LIN {X 0.305,Y -660.831,Z 854.604,A 0.000,B 0.000,C 90.000,E1 324.689} C_DIS
LIN {X -0.046,Y -663.452,Z 854.597,A 0.000,B 0.000,C 90.000,E1 323.497} C_DIS
LIN {X 0.038,Y -665.775,Z 854.590,A 0.000,B 0.000,C 90.000,E1 322.271} C_DIS
LIN {X 0.131,Y -668.429,Z 854.581,A 0.000,B 0.000,C 90.000,E1 320.561} C_DIS
LIN {X -0.225,Y -670.175,Z 854.573,A 0.000,B 0.000,C 90.000,E1 319.138} C_DIS
LIN {X -0.142,Y -671.073,Z 854.569,A 0.000,B 0.000,C 90.000,E1 318.405} C_DIS
LIN {X 0.016,Y -673.504,Z 854.558,A 0.000,B 0.000,C 90.000,E1 316.458} C_DIS
LIN {X 0.136,Y -674.995,Z 854.551,A 0.000,B 0.000,C 90.000,E1 315.243} C_DIS
LIN {X 0.192,Y -675.409,Z 854.549,A 0.000,B 0.000,C 90.000,E1 314.757} C_DIS
LIN {X -0.057,Y -677.144,Z 854.539,A 0.000,B 0.000,C 90.000,E1 313.095} C_DIS
LIN {X -0.311,Y -678.588,Z 854.531,A 0.000,B 0.000,C 90.000,E1 311.676} C_DIS
LIN {X -0.045,Y -679.939,Z 854.523,A 0.000,B 0.000,C 90.000,E1 310.216} C_DIS
LIN {X 0.327,Y -681.172,Z 854.516,A 0.000,B 0.000,C 90.000,E1 308.749} C_DIS
LIN {X -0.229,Y -682.419,Z 854.508,A 0.000,B 0.000,C 90.000,E1 307.363} C_DIS
LIN {X -0.224,Y -683.571,Z 854.500,A 0.000,B 0.000,C 90.000,E1 305.931} C_DIS
LIN {X -0.035,Y -684.565,Z 854.492,A 0.000,B 0.000,C 90.000,E1 304.485} C_DIS
LIN {X -0.013,Y -685.390,Z 854.485,A 0.000,B 0.000,C 90.000,E1 303.293} C_DIS
LIN {X 0.041,Y -686.764,Z 854.474,A 0.000,B 0.000,C 90.000,E1 301.386} C_DIS
LIN {X 0.019,Y -688.211,Z 854.464,A 0.000,B 0.000,C 90.000,E1 299.489} C_DIS
LIN {X -0.183,Y -689.701,Z 854.455,A 0.000,B 0.000,C 90.000,E1 297.847} C_DIS
LIN {X -0.206,Y -691.756,Z 854.443,A 0.000,B 0.000,C 90.000,E1 295.720} C_DIS
LIN {X -0.161,Y -692.641,Z 854.438,A 0.000,B 0.000,C 90.000,E1 294.771} C_DIS
LIN {X -0.106,Y -693.267,Z 854.432,A 0.000,B 0.000,C 90.000,E1 293.823} C_DIS
LIN {X 0.103,Y -693.192,Z 854.430,A 0.000,B 0.000,C 90.000,E1 293.334} C_DIS
LIN {X 0.345,Y -692.866,Z 854.428,A 0.000,B 0.000,C 90.000,E1 293.078} C_DIS
LIN {X -0.083,Y -691.503,Z 854.426,A 0.000,B 0.000,C 90.000,E1 292.642} C_DIS
LIN {X 0.153,Y -690.318,Z 854.424,A 0.000,B 0.000,C 90.000,E1 292.386} C_DIS
LIN {X 0.345,Y -685.933,Z 854.422,A 0.000,B 0.000,C 90.000,E1 291.897} C_DIS
LIN {X 0.197,Y -684.631,Z 854.421,A 0.000,B 0.000,C 90.000,E1 291.791} C_DIS
LIN {X -0.331,Y -682.554,Z 854.421,A 0.000,B 0.000,C 90.000,E1 291.716} C_DIS
LIN {X -0.153,Y -676.537,Z 854.419,A 0.000,B 0.000,C 90.000,E1 291.461} C_DIS
LIN {X -0.305,Y -674.797,Z 854.419,A 0.000,B 0.000,C 90.000,E1 291.408} C_DIS
LIN {X -0.113,Y -671.365,Z 854.418,A 0.000,B 0.000,C 90.000,E1 291.280} C_DIS
LIN {X 0.071,Y -666.701,Z 854.418,A 0.000,B 0.000,C 90.000,E1 291.153} C_DIS
LIN {X 0.182,Y -654.493,Z 854.416,A 0.000,B 0.000,C 90.000,E1 290.865} C_DIS
LIN {X -0.225,Y -651.097,Z 854.415,A 0.000,B 0.000,C 90.000,E1 290.791} C_DIS
LIN {X 0.006,Y -647.543,Z 854.415,A 0.000,B 0.000,C 90.000,E1 290.663} C_DIS
LIN {X -0.286,Y -642.427,Z 854.413,A 0.000,B 0.000,C 90.000,E1 290.429} C_DIS
LIN {X -0.345,Y -642.340,Z 854.413,A 0.000,B 0.000,C 90.000,E1 290.429} C_DIS
LIN {X 0.256,Y -640.659,Z 854.412,A 0.000,B 0.000,C 90.000,E1 290.174} C_DIS
LIN {X 0.212,Y -640.651,Z 854.412,A 0.000,B 0.000,C 90.000,E1 290.174} C_DIS
LIN {X 0.313,Y -640.504,Z 854.411,A 0.000,B 0.000,C 90.000,E1 289.993} C_DIS
LIN {X 0.066,Y -642.134,Z 854.409,A 0.000,B 0.000,C 90.000,E1 289.577} C_DIS
LIN {X -0.280,Y -649.483,Z 854.401,A 0.000,B 0.000,C 90.000,E1 288.236} C_DIS
LIN {X 0.093,Y -652.491,Z 854.398,A 0.000,B 0.000,C 90.000,E1 287.583} C_DIS
LIN {X -0.092,Y -655.744,Z 854.394,A 0.000,B 0.000,C 90.000,E1 286.858} C_DIS
LIN {X -0.254,Y -658.563,Z 854.390,A 0.000,B 0.000,C 90.000,E1 286.134} C_DIS
LIN {X 0.166,Y -660.214,Z 854.387,A 0.000,B 0.000,C 90.000,E1 285.607} C_DIS
LIN {X -0.131,Y -662.219,Z 854.383,A 0.000,B 0.000,C 90.000,E1 284.898} C_DIS
LIN {X -0.152,Y -663.344,Z 854.380,A 0.000,B 0.000,C 90.000,E1 284.411} C_DIS
LIN {X 0.134,Y -664.877,Z 854.375,A 0.000,B 0.000,C 90.000,E1 283.411} C_DIS
LIN {X -0.038,Y -665.424,Z 854.372,A 0.000,B 0.000,C 90.000,E1 282.939} C_DIS
LIN {X -0.351,Y -665.777,Z 854.369,A 0.000,B 0.000,C 90.000,E1 282.479} C_DIS
LIN {X 0.052,Y -665.985,Z 854.365,A 0.000,B 0.000,C 90.000,E1 281.715} C_DIS
LIN {X -0.115,Y -665.854,Z 854.362,A 0.000,B 0.000,C 90.000,E1 281.243} C_DIS
LIN {X 0.244,Y -665.514,Z 854.360,A 0.000,B 0.000,C 90.000,E1 280.725} C_DIS
LIN {X 0.071,Y -664.975,Z 854.357,A 0.000,B 0.000,C 90.000,E1 280.254} C_DIS
LIN {X -0.223,Y -664.156,Z 854.354,A 0.000,B 0.000,C 90.000,E1 279.792} C_DIS
LIN {X 0.244,Y -663.077,Z 854.352,A 0.000,B 0.000,C 90.000,E1 279.265} C_DIS
LIN {X -0.059,Y -661.694,Z 854.349,A 0.000,B 0.000,C 90.000,E1 278.803} C_DIS
LIN {X -0.270,Y -659.846,Z 854.346,A 0.000,B 0.000,C 90.000,E1 278.333} C_DIS
LIN {X 0.062,Y -657.762,Z 854.344,A 0.000,B 0.000,C 90.000,E1 277.814} C_DIS
LIN {X -0.164,Y -655.944,Z 854.341,A 0.000,B 0.000,C 90.000,E1 277.466} C_DIS
LIN {X 0.140,Y -653.194,Z 854.339,A 0.000,B 0.000,C 90.000,E1 276.947} C_DIS
LIN {X -0.186,Y -650.972,Z 854.337,A 0.000,B 0.000,C 90.000,E1 276.606} C_DIS
LIN {X 0.040,Y -646.524,Z 854.333,A 0.000,B 0.000,C 90.000,E1 275.967} C_DIS
LIN {X 0.214,Y -642.388,Z 854.330,A 0.000,B 0.000,C 90.000,E1 275.454} C_DIS
LIN {X -0.152,Y -637.498,Z 854.328,A 0.000,B 0.000,C 90.000,E1 274.992} C_DIS
LIN {X -0.286,Y -632.086,Z 854.325,A 0.000,B 0.000,C 90.000,E1 274.531} C_DIS
LIN {X 0.052,Y -624.823,Z 854.322,A 0.000,B 0.000,C 90.000,E1 273.955} C_DIS
LIN {X -0.171,Y -617.371,Z 854.319,A 0.000,B 0.000,C 90.000,E1 273.498} C_DIS
LIN {X 0.225,Y -611.014,Z 854.317,A 0.000,B 0.000,C 90.000,E1 273.094} C_DIS
LIN {X 0.111,Y -602.470,Z 854.315,A 0.000,B 0.000,C 90.000,E1 272.694} C_DIS
LIN {X 0.147,Y -597.447,Z 854.314,A 0.000,B 0.000,C 90.000,E1 272.465} C_DIS
LIN {X -0.262,Y -590.199,Z 854.312,A 0.000,B 0.000,C 90.000,E1 272.236} C_DIS
LIN {X -0.231,Y -584.532,Z 854.311,A 0.000,B 0.000,C 90.000,E1 272.064} C_DIS
LIN {X 0.037,Y -578.213,Z 854.311,A 0.000,B 0.000,C 90.000,E1 271.892} C_DIS
LIN {X 0.152,Y -571.643,Z 854.310,A 0.000,B 0.000,C 90.000,E1 271.776} C_DIS
LIN {X 0.073,Y -564.068,Z 854.310,A 0.000,B 0.000,C 90.000,E1 271.718} C_DIS
LIN {X -0.186,Y -556.079,Z 854.310,A 0.000,B 0.000,C 90.000,E1 271.718} C_DIS
LIN {X 0.047,Y -552.503,Z 854.309,A 0.000,B 0.000,C 90.000,E1 271.661} C_DIS
LIN {X 0.113,Y -549.285,Z 854.309,A 0.000,B 0.000,C 90.000,E1 271.547} C_DIS
LIN {X 0.107,Y -548.823,Z 854.308,A 0.000,B 0.000,C 90.000,E1 271.489} C_DIS
LIN {X -0.141,Y -548.111,Z 854.308,A 0.000,B 0.000,C 90.000,E1 271.375} C_DIS
LIN {X 0.206,Y -547.113,Z 854.305,A 0.000,B 0.000,C 90.000,E1 270.917} C_DIS
LIN {X -0.204,Y -546.071,Z 854.301,A 0.000,B 0.000,C 90.000,E1 270.115} C_DIS
LIN {X 0.156,Y -544.002,Z 854.286,A 0.000,B 0.000,C 90.000,E1 267.535} C_DIS
LIN {X -0.125,Y -542.650,Z 854.275,A 0.000,B 0.000,C 90.000,E1 265.584} C_DIS
LIN {X 0.127,Y -541.454,Z 854.266,A 0.000,B 0.000,C 90.000,E1 263.856} C_DIS
LIN {X -0.258,Y -540.437,Z 854.260,A 0.000,B 0.000,C 90.000,E1 262.761} C_DIS
LIN {X 0.069,Y -538.715,Z 854.249,A 0.000,B 0.000,C 90.000,E1 260.735} C_DIS
LIN {X -0.098,Y -536.794,Z 854.238,A 0.000,B 0.000,C 90.000,E1 258.757} C_DIS
LIN {X 0.196,Y -535.279,Z 854.230,A 0.000,B 0.000,C 90.000,E1 257.297} C_DIS
LIN {X 0.007,Y -533.945,Z 854.223,A 0.000,B 0.000,C 90.000,E1 256.172} C_DIS
LIN {X 0.098,Y -531.188,Z 854.210,A 0.000,B 0.000,C 90.000,E1 253.866} C_DIS
LIN {X 0.181,Y -529.507,Z 854.202,A 0.000,B 0.000,C 90.000,E1 252.417} C_DIS
LIN {X 0.244,Y -527.676,Z 854.194,A 0.000,B 0.000,C 90.000,E1 250.967} C_DIS
LIN {X 0.094,Y -526.170,Z 854.188,A 0.000,B 0.000,C 90.000,E1 249.826} C_DIS
LIN {X -0.227,Y -524.242,Z 854.180,A 0.000,B 0.000,C 90.000,E1 248.411} C_DIS
LIN {X -0.222,Y -521.671,Z 854.170,A 0.000,B 0.000,C 90.000,E1 246.666} C_DIS
LIN {X -0.092,Y -519.902,Z 854.164,A 0.000,B 0.000,C 90.000,E1 245.485} C_DIS
LIN {X 0.223,Y -518.082,Z 854.157,A 0.000,B 0.000,C 90.000,E1 244.280} C_DIS
LIN {X 0.046,Y -516.123,Z 854.151,A 0.000,B 0.000,C 90.000,E1 243.127} C_DIS
LIN {X 0.192,Y -512.528,Z 854.139,A 0.000,B 0.000,C 90.000,E1 241.051} C_DIS
LIN {X -0.167,Y -510.982,Z 854.134,A 0.000,B 0.000,C 90.000,E1 240.205} C_DIS
LIN {X 0.011,Y -507.628,Z 854.125,A 0.000,B 0.000,C 90.000,E1 238.408} C_DIS
LIN {X 0.062,Y -504.750,Z 854.116,A 0.000,B 0.000,C 90.000,E1 236.914} C_DIS
LIN {X 0.150,Y -502.887,Z 854.111,A 0.000,B 0.000,C 90.000,E1 236.008} C_DIS
LIN {X 0.101,Y -500.210,Z 854.105,A 0.000,B 0.000,C 90.000,E1 234.815} C_DIS
LIN {X 0.013,Y -497.365,Z 854.098,A 0.000,B 0.000,C 90.000,E1 233.623} C_DIS
LIN {X -0.105,Y -493.157,Z 854.088,A 0.000,B 0.000,C 90.000,E1 231.823} C_DIS
LIN {X -0.015,Y -488.793,Z 854.078,A 0.000,B 0.000,C 90.000,E1 229.989} C_DIS
LIN {X 0.093,Y -485.390,Z 854.069,A 0.000,B 0.000,C 90.000,E1 228.447} C_DIS
LIN {X -0.011,Y -479.194,Z 854.054,A 0.000,B 0.000,C 90.000,E1 225.688} C_DIS
LIN {X 0.233,Y -475.930,Z 854.045,A 0.000,B 0.000,C 90.000,E1 224.109} C_DIS
LIN {X 0.057,Y -470.544,Z 854.031,A 0.000,B 0.000,C 90.000,E1 221.634} C_DIS
LIN {X -0.111,Y -466.488,Z 854.021,A 0.000,B 0.000,C 90.000,E1 219.769} C_DIS
LIN {X 0.236,Y -463.871,Z 854.014,A 0.000,B 0.000,C 90.000,E1 218.463} C_DIS
LIN {X -0.220,Y -459.270,Z 854.002,A 0.000,B 0.000,C 90.000,E1 216.297} C_DIS
LIN {X -0.065,Y -454.412,Z 853.989,A 0.000,B 0.000,C 90.000,E1 214.040} C_DIS
LIN {X -0.094,Y -448.929,Z 853.975,A 0.000,B 0.000,C 90.000,E1 211.465} C_DIS
LIN {X -0.142,Y -443.436,Z 853.960,A 0.000,B 0.000,C 90.000,E1 208.871} C_DIS
LIN {X 0.082,Y -440.075,Z 853.951,A 0.000,B 0.000,C 90.000,E1 207.206} C_DIS
LIN {X -0.149,Y -436.707,Z 853.942,A 0.000,B 0.000,C 90.000,E1 205.591} C_DIS
LIN {X -0.023,Y -432.647,Z 853.931,A 0.000,B 0.000,C 90.000,E1 203.590} C_DIS
LIN {X 0.004,Y -428.619,Z 853.920,A 0.000,B 0.000,C 90.000,E1 201.589} C_DIS
LIN {X 0.020,Y -426.021,Z 853.913,A 0.000,B 0.000,C 90.000,E1 200.248} C_DIS
LIN {X 0.149,Y -421.439,Z 853.899,A 0.000,B 0.000,C 90.000,E1 197.873} C_DIS
LIN {X -0.038,Y -418.215,Z 853.890,A 0.000,B 0.000,C 90.000,E1 196.205} C_DIS
LIN {X -0.074,Y -416.086,Z 853.884,A 0.000,B 0.000,C 90.000,E1 195.190} C_DIS
LIN {X -0.103,Y -413.280,Z 853.877,A 0.000,B 0.000,C 90.000,E1 193.828} C_DIS
LIN {X 0.018,Y -407.250,Z 853.860,A 0.000,B 0.000,C 90.000,E1 190.715} C_DIS
LIN {X 0.083,Y -403.143,Z 853.848,A 0.000,B 0.000,C 90.000,E1 188.624} C_DIS
LIN {X -0.057,Y -399.072,Z 853.836,A 0.000,B 0.000,C 90.000,E1 186.549} C_DIS
LIN {X -0.128,Y -392.992,Z 853.817,A 0.000,B 0.000,C 90.000,E1 183.037} C_DIS
LIN {X 0.111,Y -389.410,Z 853.803,A 0.000,B 0.000,C 90.000,E1 180.516} C_DIS
LIN {X 0.050,Y -386.974,Z 853.793,A 0.000,B 0.000,C 90.000,E1 178.740} C_DIS
LIN {X -0.143,Y -383.971,Z 853.781,A 0.000,B 0.000,C 90.000,E1 176.617} C_DIS
LIN {X 0.096,Y -381.531,Z 853.771,A 0.000,B 0.000,C 90.000,E1 174.780} C_DIS
LIN {X 0.013,Y -377.867,Z 853.755,A 0.000,B 0.000,C 90.000,E1 171.894} C_DIS
LIN {X 0.064,Y -372.888,Z 853.725,A 0.000,B 0.000,C 90.000,E1 166.408} C_DIS
LIN {X 0.059,Y -372.070,Z 853.714,A 0.000,B 0.000,C 90.000,E1 164.574} C_DIS
LIN {X 0.138,Y -372.143,Z 853.704,A 0.000,B 0.000,C 90.000,E1 162.725} C_DIS
LIN {X 0.072,Y -372.712,Z 853.700,A 0.000,B 0.000,C 90.000,E1 162.000} C_DIS
LIN {X -0.017,Y -374.058,Z 853.694,A 0.000,B 0.000,C 90.000,E1 160.913} C_DIS
LIN {X -0.010,Y -374.593,Z 853.693,A 0.000,B 0.000,C 90.000,E1 160.678} C_DIS
LIN {X 0.068,Y -375.876,Z 853.689,A 0.000,B 0.000,C 90.000,E1 159.934} C_DIS
LIN {X 0.047,Y -376.938,Z 853.687,A 0.000,B 0.000,C 90.000,E1 159.571} C_DIS
LIN {X 0.132,Y -378.868,Z 853.684,A 0.000,B 0.000,C 90.000,E1 159.028} C_DIS
LIN {X 0.124,Y -379.696,Z 853.683,A 0.000,B 0.000,C 90.000,E1 158.847} C_DIS
LIN {X -0.100,Y -384.318,Z 853.679,A 0.000,B 0.000,C 90.000,E1 158.156} C_DIS
LIN {X 0.155,Y -385.649,Z 853.678,A 0.000,B 0.000,C 90.000,E1 157.975} C_DIS
LIN {X -0.074,Y -390.628,Z 853.675,A 0.000,B 0.000,C 90.000,E1 157.592} C_DIS
LIN {X -0.108,Y -392.245,Z 853.675,A 0.000,B 0.000,C 90.000,E1 157.486} C_DIS
LIN {X 0.020,Y -398.045,Z 853.673,A 0.000,B 0.000,C 90.000,E1 157.177} C_DIS
LIN {X -0.120,Y -408.863,Z 853.671,A 0.000,B 0.000,C 90.000,E1 156.741} C_DIS
LIN {X -0.192,Y -415.764,Z 853.669,A 0.000,B 0.000,C 90.000,E1 156.485} C_DIS
LIN {X -0.146,Y -422.411,Z 853.668,A 0.000,B 0.000,C 90.000,E1 156.177} C_DIS
LIN {X -0.191,Y -430.182,Z 853.665,A 0.000,B 0.000,C 90.000,E1 155.741} C_DIS
LIN {X -0.154,Y -438.432,Z 853.662,A 0.000,B 0.000,C 90.000,E1 155.229} C_DIS
LIN {X 0.170,Y -447.724,Z 853.659,A 0.000,B 0.000,C 90.000,E1 154.537} C_DIS
LIN {X 0.036,Y -458.604,Z 853.654,A 0.000,B 0.000,C 90.000,E1 153.691} C_DIS
LIN {X -0.049,Y -464.301,Z 853.651,A 0.000,B 0.000,C 90.000,E1 153.179} C_DIS
LIN {X -0.045,Y -469.880,Z 853.648,A 0.000,B 0.000,C 90.000,E1 152.615} C_DIS
LIN {X -0.010,Y -475.194,Z 853.645,A 0.000,B 0.000,C 90.000,E1 152.025} C_DIS
LIN {X -0.089,Y -484.388,Z 853.639,A 0.000,B 0.000,C 90.000,E1 151.001} C_DIS
LIN {X -0.014,Y -492.068,Z 853.634,A 0.000,B 0.000,C 90.000,E1 150.078} C_DIS
LIN {X 0.097,Y -499.047,Z 853.629,A 0.000,B 0.000,C 90.000,E1 149.154} C_DIS
LIN {X -0.009,Y -502.452,Z 853.626,A 0.000,B 0.000,C 90.000,E1 148.742} C_DIS
LIN {X -0.212,Y -509.109,Z 853.621,A 0.000,B 0.000,C 90.000,E1 147.867} C_DIS
LIN {X 0.286,Y -517.023,Z 853.615,A 0.000,B 0.000,C 90.000,E1 146.628} C_DIS
LIN {X -0.021,Y -521.485,Z 853.611,A 0.000,B 0.000,C 90.000,E1 145.928} C_DIS
LIN {X 0.109,Y -527.451,Z 853.605,A 0.000,B 0.000,C 90.000,E1 144.895} C_DIS
LIN {X -0.108,Y -531.445,Z 853.601,A 0.000,B 0.000,C 90.000,E1 144.196} C_DIS
LIN {X 0.087,Y -543.109,Z 853.589,A 0.000,B 0.000,C 90.000,E1 142.029} C_DIS
LIN {X -0.091,Y -552.534,Z 853.580,A 0.000,B 0.000,C 90.000,E1 140.356} C_DIS
LIN {X 0.031,Y -555.668,Z 853.577,A 0.000,B 0.000,C 90.000,E1 139.784} C_DIS
LIN {X 0.081,Y -562.213,Z 853.570,A 0.000,B 0.000,C 90.000,E1 138.528} C_DIS
LIN {X -0.024,Y -570.218,Z 853.561,A 0.000,B 0.000,C 90.000,E1 137.025} C_DIS
LIN {X 0.140,Y -574.938,Z 853.556,A 0.000,B 0.000,C 90.000,E1 136.053} C_DIS
LIN {X -0.175,Y -580.233,Z 853.550,A 0.000,B 0.000,C 90.000,E1 135.000} C_DIS
LIN {X 0.000,Y -585.465,Z 853.544,A 0.000,B 0.000,C 90.000,E1 133.905} C_DIS
LIN {X -0.065,Y -589.929,Z 853.539,A 0.000,B 0.000,C 90.000,E1 132.975} C_DIS
LIN {X 0.178,Y -592.991,Z 853.535,A 0.000,B 0.000,C 90.000,E1 132.285} C_DIS
LIN {X -0.098,Y -598.779,Z 853.528,A 0.000,B 0.000,C 90.000,E1 130.987} C_DIS
LIN {X 0.179,Y -604.404,Z 853.520,A 0.000,B 0.000,C 90.000,E1 129.644} C_DIS
LIN {X -0.033,Y -605.514,Z 853.519,A 0.000,B 0.000,C 90.000,E1 129.402} C_DIS
LIN {X -0.025,Y -610.395,Z 853.512,A 0.000,B 0.000,C 90.000,E1 128.096} C_DIS
LIN {X -0.029,Y -613.075,Z 853.507,A 0.000,B 0.000,C 90.000,E1 127.317} C_DIS
LIN {X 0.001,Y -615.649,Z 853.503,A 0.000,B 0.000,C 90.000,E1 126.537} C_DIS
LIN {X 0.180,Y -619.642,Z 853.496,A 0.000,B 0.000,C 90.000,E1 125.231} C_DIS
LIN {X -0.298,Y -623.002,Z 853.489,A 0.000,B 0.000,C 90.000,E1 123.992} C_DIS
LIN {X -0.189,Y -625.312,Z 853.483,A 0.000,B 0.000,C 90.000,E1 122.959} C_DIS
LIN {X -0.390,Y -626.894,Z 853.479,A 0.000,B 0.000,C 90.000,E1 122.212} C_DIS
LIN {X 0.298,Y -628.727,Z 853.473,A 0.000,B 0.000,C 90.000,E1 121.131} C_DIS
LIN {X 0.196,Y -631.203,Z 853.465,A 0.000,B 0.000,C 90.000,E1 119.617} C_DIS
LIN {X 0.040,Y -632.158,Z 853.460,A 0.000,B 0.000,C 90.000,E1 118.871} C_DIS
LIN {X 0.141,Y -633.050,Z 853.456,A 0.000,B 0.000,C 90.000,E1 118.103} C_DIS
LIN {X -0.267,Y -633.921,Z 853.451,A 0.000,B 0.000,C 90.000,E1 117.129} C_DIS
LIN {X -0.185,Y -634.207,Z 853.448,A 0.000,B 0.000,C 90.000,E1 116.616} C_DIS
LIN {X -0.017,Y -634.318,Z 853.442,A 0.000,B 0.000,C 90.000,E1 115.591} C_DIS
LIN {X 0.025,Y -634.254,Z 853.441,A 0.000,B 0.000,C 90.000,E1 115.335} C_DIS
LIN {X -0.078,Y -633.499,Z 853.435,A 0.000,B 0.000,C 90.000,E1 114.335} C_DIS
LIN {X -0.003,Y -632.746,Z 853.432,A 0.000,B 0.000,C 90.000,E1 113.823} C_DIS
LIN {X -0.188,Y -631.298,Z 853.430,A 0.000,B 0.000,C 90.000,E1 113.334} C_DIS
LIN {X -0.157,Y -630.372,Z 853.428,A 0.000,B 0.000,C 90.000,E1 113.078} C_DIS
LIN {X -0.144,Y -629.516,Z 853.427,A 0.000,B 0.000,C 90.000,E1 112.950} C_DIS
LIN {X -0.353,Y -627.650,Z 853.425,A 0.000,B 0.000,C 90.000,E1 112.589} C_DIS
LIN {X -0.344,Y -626.450,Z 853.425,A 0.000,B 0.000,C 90.000,E1 112.461} C_DIS
LIN {X 0.250,Y -623.409,Z 853.423,A 0.000,B 0.000,C 90.000,E1 112.025} C_DIS
LIN {X 0.248,Y -620.100,Z 853.421,A 0.000,B 0.000,C 90.000,E1 111.770} C_DIS
LIN {X 0.026,Y -617.046,Z 853.420,A 0.000,B 0.000,C 90.000,E1 111.535} C_DIS
LIN {X -0.217,Y -610.855,Z 853.417,A 0.000,B 0.000,C 90.000,E1 111.153} C_DIS
LIN {X -0.223,Y -601.454,Z 853.414,A 0.000,B 0.000,C 90.000,E1 110.610} C_DIS
LIN {X -0.157,Y -594.867,Z 853.412,A 0.000,B 0.000,C 90.000,E1 110.248} C_DIS
LIN {X 0.163,Y -588.110,Z 853.411,A 0.000,B 0.000,C 90.000,E1 109.885} C_DIS
LIN {X -0.289,Y -579.028,Z 853.409,A 0.000,B 0.000,C 90.000,E1 109.577} C_DIS
LIN {X -0.286,Y -574.865,Z 853.408,A 0.000,B 0.000,C 90.000,E1 109.450} C_DIS
LIN {X 0.034,Y -567.390,Z 853.406,A 0.000,B 0.000,C 90.000,E1 109.141} C_DIS
LIN {X -0.054,Y -566.248,Z 853.406,A 0.000,B 0.000,C 90.000,E1 109.087} C_DIS
LIN {X -0.125,Y -564.156,Z 853.405,A 0.000,B 0.000,C 90.000,E1 108.906} C_DIS
LIN {X -0.220,Y -562.671,Z 853.404,A 0.000,B 0.000,C 90.000,E1 108.671} C_DIS
LIN {X 0.137,Y -561.346,Z 853.401,A 0.000,B 0.000,C 90.000,E1 108.236} C_DIS
LIN {X 0.160,Y -560.574,Z 853.399,A 0.000,B 0.000,C 90.000,E1 107.819} C_DIS
LIN {X 0.251,Y -560.171,Z 853.394,A 0.000,B 0.000,C 90.000,E1 106.858} C_DIS
LIN {X -0.233,Y -561.442,Z 853.369,A 0.000,B 0.000,C 90.000,E1 102.479} C_DIS
LIN {X -0.084,Y -562.863,Z 853.357,A 0.000,B 0.000,C 90.000,E1 100.254} C_DIS
LIN {X 0.063,Y -563.850,Z 853.349,A 0.000,B 0.000,C 90.000,E1 98.859} C_DIS
LIN {X 0.147,Y -564.822,Z 853.342,A 0.000,B 0.000,C 90.000,E1 97.473} C_DIS
LIN {X -0.153,Y -565.751,Z 853.332,A 0.000,B 0.000,C 90.000,E1 95.853} C_DIS
LIN {X 0.009,Y -566.515,Z 853.323,A 0.000,B 0.000,C 90.000,E1 94.188} C_DIS
LIN {X 0.077,Y -567.024,Z 853.316,A 0.000,B 0.000,C 90.000,E1 92.808} C_DIS
LIN {X 0.115,Y -567.401,Z 853.308,A 0.000,B 0.000,C 90.000,E1 91.432} C_DIS
LIN {X 0.150,Y -567.795,Z 853.300,A 0.000,B 0.000,C 90.000,E1 90.057} C_DIS
LIN {X -0.116,Y -568.222,Z 853.290,A 0.000,B 0.000,C 90.000,E1 88.165} C_DIS
LIN {X -0.046,Y -568.481,Z 853.282,A 0.000,B 0.000,C 90.000,E1 86.788} C_DIS
LIN {X -0.271,Y -568.784,Z 853.272,A 0.000,B 0.000,C 90.000,E1 84.894} C_DIS
LIN {X 0.181,Y -569.162,Z 853.261,A 0.000,B 0.000,C 90.000,E1 82.932} C_DIS
LIN {X 0.255,Y -569.724,Z 853.249,A 0.000,B 0.000,C 90.000,E1 80.735} C_DIS
LIN {X -0.226,Y -570.394,Z 853.238,A 0.000,B 0.000,C 90.000,E1 78.870} C_DIS
LIN {X 0.162,Y -570.899,Z 853.231,A 0.000,B 0.000,C 90.000,E1 77.465} C_DIS
LIN {X 0.183,Y -571.500,Z 853.221,A 0.000,B 0.000,C 90.000,E1 75.825} C_DIS
LIN {X -0.057,Y -571.829,Z 853.212,A 0.000,B 0.000,C 90.000,E1 74.212} C_DIS
LIN {X -0.261,Y -572.057,Z 853.206,A 0.000,B 0.000,C 90.000,E1 73.142} C_DIS
LIN {X 0.233,Y -572.207,Z 853.197,A 0.000,B 0.000,C 90.000,E1 71.456} C_DIS
LIN {X 0.000,Y -572.114,Z 853.187,A 0.000,B 0.000,C 90.000,E1 69.571} C_DIS
LIN {X -0.038,Y -572.013,Z 853.176,A 0.000,B 0.000,C 90.000,E1 67.667} C_DIS
LIN {X -0.224,Y -571.890,Z 853.167,A 0.000,B 0.000,C 90.000,E1 66.049} C_DIS
LIN {X -0.183,Y -571.460,Z 853.158,A 0.000,B 0.000,C 90.000,E1 64.409} C_DIS
LIN {X 0.263,Y -571.013,Z 853.150,A 0.000,B 0.000,C 90.000,E1 62.999} C_DIS
LIN {X -0.141,Y -570.683,Z 853.144,A 0.000,B 0.000,C 90.000,E1 61.948} C_DIS
LIN {X -0.214,Y -569.975,Z 853.137,A 0.000,B 0.000,C 90.000,E1 60.589} C_DIS
LIN {X 0.040,Y -569.518,Z 853.132,A 0.000,B 0.000,C 90.000,E1 59.744} C_DIS
LIN {X -0.095,Y -568.553,Z 853.126,A 0.000,B 0.000,C 90.000,E1 58.663} C_DIS
LIN {X -0.239,Y -567.541,Z 853.120,A 0.000,B 0.000,C 90.000,E1 57.582} C_DIS
LIN {X 0.072,Y -566.249,Z 853.114,A 0.000,B 0.000,C 90.000,E1 56.453} C_DIS
LIN {X -0.267,Y -564.748,Z 853.108,A 0.000,B 0.000,C 90.000,E1 55.388} C_DIS
LIN {X 0.063,Y -563.506,Z 853.103,A 0.000,B 0.000,C 90.000,E1 54.529} C_DIS
LIN {X 0.052,Y -562.145,Z 853.098,A 0.000,B 0.000,C 90.000,E1 53.703} C_DIS
LIN {X 0.005,Y -560.021,Z 853.092,A 0.000,B 0.000,C 90.000,E1 52.603} C_DIS
LIN {X -0.148,Y -558.887,Z 853.089,A 0.000,B 0.000,C 90.000,E1 52.065} C_DIS
LIN {X -0.324,Y -556.910,Z 853.085,A 0.000,B 0.000,C 90.000,E1 51.251} C_DIS
LIN {X 0.264,Y -554.683,Z 853.080,A 0.000,B 0.000,C 90.000,E1 50.356} C_DIS
LIN {X 0.046,Y -552.157,Z 853.075,A 0.000,B 0.000,C 90.000,E1 49.542} C_DIS
LIN {X -0.254,Y -550.320,Z 853.072,A 0.000,B 0.000,C 90.000,E1 49.013} C_DIS
LIN {X -0.118,Y -546.034,Z 853.066,A 0.000,B 0.000,C 90.000,E1 47.877} C_DIS
LIN {X -0.092,Y -543.710,Z 853.063,A 0.000,B 0.000,C 90.000,E1 47.310} C_DIS
LIN {X -0.077,Y -541.190,Z 853.060,A 0.000,B 0.000,C 90.000,E1 46.743} C_DIS
LIN {X -0.271,Y -537.690,Z 853.056,A 0.000,B 0.000,C 90.000,E1 46.053} C_DIS
LIN {X 0.277,Y -535.515,Z 853.053,A 0.000,B 0.000,C 90.000,E1 45.567} C_DIS
LIN {X 0.023,Y -531.380,Z 853.049,A 0.000,B 0.000,C 90.000,E1 44.879} C_DIS
LIN {X 0.321,Y -527.825,Z 853.046,A 0.000,B 0.000,C 90.000,E1 44.271} C_DIS
LIN {X 0.216,Y -523.953,Z 853.043,A 0.000,B 0.000,C 90.000,E1 43.704} C_DIS
LIN {X 0.030,Y -518.799,Z 853.039,A 0.000,B 0.000,C 90.000,E1 43.014} C_DIS
LIN {X -0.276,Y -515.440,Z 853.037,A 0.000,B 0.000,C 90.000,E1 42.609} C_DIS
LIN {X -0.089,Y -510.649,Z 853.033,A 0.000,B 0.000,C 90.000,E1 42.000} C_DIS
LIN {X 0.181,Y -504.272,Z 853.029,A 0.000,B 0.000,C 90.000,E1 41.229} C_DIS
LIN {X -0.268,Y -498.876,Z 853.026,A 0.000,B 0.000,C 90.000,E1 40.701} C_DIS
LIN {X 0.110,Y -493.308,Z 853.023,A 0.000,B 0.000,C 90.000,E1 40.092} C_DIS
LIN {X 0.083,Y -487.671,Z 853.020,A 0.000,B 0.000,C 90.000,E1 39.564} C_DIS
LIN {X -0.247,Y -478.976,Z 853.016,A 0.000,B 0.000,C 90.000,E1 38.830} C_DIS
LIN {X 0.239,Y -469.819,Z 853.011,A 0.000,B 0.000,C 90.000,E1 38.016} C_DIS
LIN {X 0.244,Y -458.891,Z 853.007,A 0.000,B 0.000,C 90.000,E1 37.156} C_DIS
LIN {X 0.121,Y -444.804,Z 853.001,A 0.000,B 0.000,C 90.000,E1 36.091} C_DIS
LIN {X 0.068,Y -419.930,Z 852.990,A 0.000,B 0.000,C 90.000,E1 34.119} C_DIS
LIN {X 0.141,Y -403.547,Z 852.981,A 0.000,B 0.000,C 90.000,E1 32.625} C_DIS
LIN {X -0.165,Y -398.705,Z 852.978,A 0.000,B 0.000,C 90.000,E1 32.133} C_DIS
LIN {X -0.033,Y -395.347,Z 852.976,A 0.000,B 0.000,C 90.000,E1 31.671} C_DIS
LIN {X 0.055,Y -393.645,Z 852.974,A 0.000,B 0.000,C 90.000,E1 31.386} C_DIS
LIN {X 0.099,Y -392.794,Z 852.974,A 0.000,B 0.000,C 90.000,E1 31.209} C_DIS
LIN {X 0.010,Y -392.267,Z 852.973,A 0.000,B 0.000,C 90.000,E1 31.052} C_DIS
LIN {X -0.079,Y -390.365,Z 852.967,A 0.000,B 0.000,C 90.000,E1 30.001} C_DIS
LIN {X -0.038,Y -390.119,Z 852.964,A 0.000,B 0.000,C 90.000,E1 29.461} C_DIS
LIN {X 0.188,Y -390.290,Z 852.958,A 0.000,B 0.000,C 90.000,E1 28.359} C_DIS
LIN {X 0.000,Y -392.051,Z 852.942,A 0.000,B 0.000,C 90.000,E1 25.540} C_DIS
LIN {X -0.151,Y -393.977,Z 852.928,A 0.000,B 0.000,C 90.000,E1 23.078} C_DIS
LIN {X 0.111,Y -395.859,Z 852.916,A 0.000,B 0.000,C 90.000,E1 20.918} C_DIS
LIN {X -0.099,Y -397.950,Z 852.905,A 0.000,B 0.000,C 90.000,E1 18.833} C_DIS
LIN {X -0.145,Y -400.314,Z 852.893,A 0.000,B 0.000,C 90.000,E1 16.732} C_DIS
LIN {X 0.131,Y -403.421,Z 852.879,A 0.000,B 0.000,C 90.000,E1 14.245} C_DIS
LIN {X 0.010,Y -406.959,Z 852.866,A 0.000,B 0.000,C 90.000,E1 11.827} C_DIS
LIN {X 0.189,Y -410.276,Z 852.854,A 0.000,B 0.000,C 90.000,E1 9.726} C_DIS
LIN {X -0.053,Y -414.319,Z 852.841,A 0.000,B 0.000,C 90.000,E1 7.352} C_DIS
LIN {X 0.136,Y -418.615,Z 852.828,A 0.000,B 0.000,C 90.000,E1 4.935} C_DIS
LIN {X 0.150,Y -425.355,Z 852.809,A 0.000,B 0.000,C 90.000,E1 1.547} C_DIS
LIN {X -0.197,Y -430.076,Z 852.797,A 0.000,B 0.000,C 90.000,E1 359.484} C_DIS
LIN {X -0.055,Y -435.683,Z 852.784,A 0.000,B 0.000,C 90.000,E1 357.135} C_DIS
LIN {X 0.046,Y -439.834,Z 852.775,A 0.000,B 0.000,C 90.000,E1 355.469} C_DIS
LIN {X -0.170,Y -444.240,Z 852.766,A 0.000,B 0.000,C 90.000,E1 353.856} C_DIS
LIN {X 0.053,Y -445.823,Z 852.763,A 0.000,B 0.000,C 90.000,E1 353.337} C_DIS
LIN {X -0.157,Y -447.822,Z 852.760,A 0.000,B 0.000,C 90.000,E1 352.875} C_DIS
LIN {X 0.092,Y -450.075,Z 852.758,A 0.000,B 0.000,C 90.000,E1 352.470} C_DIS
LIN {X -0.160,Y -452.668,Z 852.757,A 0.000,B 0.000,C 90.000,E1 352.186} C_DIS
LIN {X -0.227,Y -457.969,Z 852.754,A 0.000,B 0.000,C 90.000,E1 351.781} C_DIS
LIN {X -0.129,Y -470.002,Z 852.751,A 0.000,B 0.000,C 90.000,E1 351.141} C_DIS
LIN {X -0.034,Y -476.721,Z 852.749,A 0.000,B 0.000,C 90.000,E1 350.792} C_DIS
LIN {X -0.195,Y -486.471,Z 852.746,A 0.000,B 0.000,C 90.000,E1 350.274} C_DIS
LIN {X -0.154,Y -496.057,Z 852.743,A 0.000,B 0.000,C 90.000,E1 349.690} C_DIS
LIN {X -0.086,Y -508.609,Z 852.738,A 0.000,B 0.000,C 90.000,E1 348.870} C_DIS
LIN {X -0.084,Y -516.418,Z 852.735,A 0.000,B 0.000,C 90.000,E1 348.342} C_DIS
LIN {X 0.292,Y -524.086,Z 852.732,A 0.000,B 0.000,C 90.000,E1 347.757} C_DIS
LIN {X -0.084,Y -530.094,Z 852.730,A 0.000,B 0.000,C 90.000,E1 347.353} C_DIS
LIN {X 0.086,Y -540.376,Z 852.725,A 0.000,B 0.000,C 90.000,E1 346.520} C_DIS
LIN {X -0.067,Y -546.070,Z 852.723,A 0.000,B 0.000,C 90.000,E1 346.061} C_DIS
LIN {X 0.301,Y -554.189,Z 852.718,A 0.000,B 0.000,C 90.000,E1 345.283} C_DIS
LIN {X 0.180,Y -562.131,Z 852.714,A 0.000,B 0.000,C 90.000,E1 344.519} C_DIS
LIN {X -0.017,Y -568.316,Z 852.710,A 0.000,B 0.000,C 90.000,E1 343.866} C_DIS
LIN {X 0.115,Y -575.502,Z 852.706,A 0.000,B 0.000,C 90.000,E1 343.032} C_DIS
LIN {X 0.154,Y -584.026,Z 852.700,A 0.000,B 0.000,C 90.000,E1 341.945} C_DIS
LIN {X 0.151,Y -588.869,Z 852.696,A 0.000,B 0.000,C 90.000,E1 341.275} C_DIS
LIN {X 0.192,Y -593.331,Z 852.692,A 0.000,B 0.000,C 90.000,E1 340.604} C_DIS
LIN {X 0.275,Y -597.516,Z 852.689,A 0.000,B 0.000,C 90.000,E1 339.934} C_DIS
LIN {X 0.139,Y -602.378,Z 852.684,A 0.000,B 0.000,C 90.000,E1 339.156} C_DIS
LIN {X 0.167,Y -609.113,Z 852.678,A 0.000,B 0.000,C 90.000,E1 337.975} C_DIS
LIN {X -0.226,Y -614.105,Z 852.673,A 0.000,B 0.000,C 90.000,E1 337.102} C_DIS
LIN {X 0.012,Y -618.149,Z 852.668,A 0.000,B 0.000,C 90.000,E1 336.305} C_DIS
LIN {X -0.028,Y -622.679,Z 852.663,A 0.000,B 0.000,C 90.000,E1 335.409} C_DIS
LIN {X -0.269,Y -627.475,Z 852.658,A 0.000,B 0.000,C 90.000,E1 334.409} C_DIS
LIN {X -0.185,Y -632.031,Z 852.652,A 0.000,B 0.000,C 90.000,E1 333.384} C_DIS
LIN {X 0.004,Y -637.136,Z 852.645,A 0.000,B 0.000,C 90.000,E1 332.103} C_DIS
LIN {X 0.019,Y -641.927,Z 852.638,A 0.000,B 0.000,C 90.000,E1 330.845} C_DIS
LIN {X 0.214,Y -644.744,Z 852.634,A 0.000,B 0.000,C 90.000,E1 330.078} C_DIS
LIN {X 0.276,Y -648.232,Z 852.628,A 0.000,B 0.000,C 90.000,E1 329.076} C_DIS
LIN {X -0.168,Y -651.494,Z 852.623,A 0.000,B 0.000,C 90.000,E1 328.122} C_DIS
LIN {X 0.428,Y -655.154,Z 852.616,A 0.000,B 0.000,C 90.000,E1 326.834} C_DIS
LIN {X 0.072,Y -657.869,Z 852.611,A 0.000,B 0.000,C 90.000,E1 325.881} C_DIS
LIN {X 0.119,Y -660.315,Z 852.605,A 0.000,B 0.000,C 90.000,E1 324.895} C_DIS
LIN {X -0.238,Y -663.043,Z 852.598,A 0.000,B 0.000,C 90.000,E1 323.703} C_DIS
LIN {X -0.160,Y -665.479,Z 852.591,A 0.000,B 0.000,C 90.000,E1 322.477} C_DIS
LIN {X -0.043,Y -667.422,Z 852.585,A 0.000,B 0.000,C 90.000,E1 321.251} C_DIS
LIN {X 0.018,Y -668.602,Z 852.581,A 0.000,B 0.000,C 90.000,E1 320.517} C_DIS
LIN {X 0.092,Y -670.377,Z 852.573,A 0.000,B 0.000,C 90.000,E1 319.057} C_DIS
LIN {X 0.188,Y -671.557,Z 852.567,A 0.000,B 0.000,C 90.000,E1 318.081} C_DIS
LIN {X -0.166,Y -673.475,Z 852.559,A 0.000,B 0.000,C 90.000,E1 316.662} C_DIS
LIN {X 0.391,Y -674.369,Z 852.555,A 0.000,B 0.000,C 90.000,E1 315.891} C_DIS
LIN {X 0.416,Y -674.595,Z 852.554,A 0.000,B 0.000,C 90.000,E1 315.648} C_DIS
LIN {X -0.031,Y -674.990,Z 852.552,A 0.000,B 0.000,C 90.000,E1 315.445} C_DIS
LIN {X 0.021,Y -675.368,Z 852.550,A 0.000,B 0.000,C 90.000,E1 314.960} C_DIS
LIN {X -0.398,Y -675.903,Z 852.547,A 0.000,B 0.000,C 90.000,E1 314.514} C_DIS
LIN {X 0.286,Y -677.414,Z 852.539,A 0.000,B 0.000,C 90.000,E1 313.014} C_DIS
LIN {X 0.035,Y -678.870,Z 852.531,A 0.000,B 0.000,C 90.000,E1 311.595} C_DIS
LIN {X -0.133,Y -680.207,Z 852.523,A 0.000,B 0.000,C 90.000,E1 310.172} C_DIS
LIN {X -0.275,Y -681.467,Z 852.515,A 0.000,B 0.000,C 90.000,E1 308.749} C_DIS
LIN {X 0.102,Y -682.516,Z 852.509,A 0.000,B 0.000,C 90.000,E1 307.523} C_DIS
LIN {X 0.117,Y -683.690,Z 852.501,A 0.000,B 0.000,C 90.000,E1 306.091} C_DIS
LIN {X 0.129,Y -684.540,Z 852.494,A 0.000,B 0.000,C 90.000,E1 304.898} C_DIS
LIN {X -0.224,Y -685.525,Z 852.486,A 0.000,B 0.000,C 90.000,E1 303.499} C_DIS
LIN {X -0.163,Y -686.874,Z 852.475,A 0.000,B 0.000,C 90.000,E1 301.592} C_DIS
LIN {X 0.160,Y -688.325,Z 852.465,A 0.000,B 0.000,C 90.000,E1 299.667} C_DIS
LIN {X 0.182,Y -689.983,Z 852.454,A 0.000,B 0.000,C 90.000,E1 297.769} C_DIS
LIN {X -0.083,Y -691.772,Z 852.444,A 0.000,B 0.000,C 90.000,E1 295.899} C_DIS
LIN {X -0.090,Y -692.873,Z 852.437,A 0.000,B 0.000,C 90.000,E1 294.719} C_DIS
LIN {X 0.010,Y -693.360,Z 852.433,A 0.000,B 0.000,C 90.000,E1 294.003} C_DIS
LIN {X 0.216,Y -693.390,Z 852.431,A 0.000,B 0.000,C 90.000,E1 293.515} C_DIS
LIN {X 0.184,Y -693.325,Z 852.430,A 0.000,B 0.000,C 90.000,E1 293.281} C_DIS
LIN {X -0.209,Y -692.891,Z 852.428,A 0.000,B 0.000,C 90.000,E1 293.078} C_DIS
LIN {X 0.031,Y -692.210,Z 852.427,A 0.000,B 0.000,C 90.000,E1 292.823} C_DIS
LIN {X 0.003,Y -691.374,Z 852.426,A 0.000,B 0.000,C 90.000,E1 292.589} C_DIS
LIN {X 0.121,Y -690.828,Z 852.425,A 0.000,B 0.000,C 90.000,E1 292.461} C_DIS
LIN {X 0.239,Y -689.988,Z 852.424,A 0.000,B 0.000,C 90.000,E1 292.333} C_DIS
LIN {X -0.318,Y -686.607,Z 852.422,A 0.000,B 0.000,C 90.000,E1 292.025} C_DIS
LIN {X -0.207,Y -685.306,Z 852.422,A 0.000,B 0.000,C 90.000,E1 291.897} C_DIS
LIN {X -0.038,Y -683.826,Z 852.421,A 0.000,B 0.000,C 90.000,E1 291.770} C_DIS
LIN {X -0.122,Y -681.458,Z 852.420,A 0.000,B 0.000,C 90.000,E1 291.663} C_DIS
LIN {X 0.203,Y -677.434,Z 852.419,A 0.000,B 0.000,C 90.000,E1 291.482} C_DIS
LIN {X -0.340,Y -674.209,Z 852.419,A 0.000,B 0.000,C 90.000,E1 291.408} C_DIS
LIN {X 0.305,Y -670.132,Z 852.418,A 0.000,B 0.000,C 90.000,E1 291.227} C_DIS
LIN {X -0.055,Y -654.812,Z 852.416,A 0.000,B 0.000,C 90.000,E1 290.918} C_DIS
LIN {X 0.142,Y -648.696,Z 852.415,A 0.000,B 0.000,C 90.000,E1 290.737} C_DIS
LIN {X -0.095,Y -646.269,Z 852.415,A 0.000,B 0.000,C 90.000,E1 290.663} C_DIS
LIN {X -0.161,Y -641.453,Z 852.413,A 0.000,B 0.000,C 90.000,E1 290.429} C_DIS
LIN {X -0.233,Y -639.416,Z 852.412,A 0.000,B 0.000,C 90.000,E1 290.248} C_DIS
LIN {X 0.105,Y -639.127,Z 852.412,A 0.000,B 0.000,C 90.000,E1 290.194} C_DIS
LIN {X 0.061,Y -639.080,Z 852.412,A 0.000,B 0.000,C 90.000,E1 290.194} C_DIS
LIN {X -0.311,Y -639.016,Z 852.411,A 0.000,B 0.000,C 90.000,E1 290.066} C_DIS
LIN {X -0.012,Y -640.226,Z 852.409,A 0.000,B 0.000,C 90.000,E1 289.685} C_DIS
LIN {X -0.261,Y -642.688,Z 852.407,A 0.000,B 0.000,C 90.000,E1 289.214} C_DIS
LIN {X 0.105,Y -647.472,Z 852.402,A 0.000,B 0.000,C 90.000,E1 288.308} C_DIS
LIN {X -0.091,Y -651.644,Z 852.397,A 0.000,B 0.000,C 90.000,E1 287.457} C_DIS
LIN {X -0.163,Y -653.832,Z 852.394,A 0.000,B 0.000,C 90.000,E1 286.968} C_DIS
LIN {X 0.099,Y -656.713,Z 852.390,A 0.000,B 0.000,C 90.000,E1 286.205} C_DIS
LIN {X 0.054,Y -658.411,Z 852.387,A 0.000,B 0.000,C 90.000,E1 285.717} C_DIS
LIN {X -0.265,Y -660.532,Z 852.383,A 0.000,B 0.000,C 90.000,E1 285.009} C_DIS
LIN {X 0.177,Y -661.687,Z 852.381,A 0.000,B 0.000,C 90.000,E1 284.481} C_DIS
LIN {X -0.104,Y -662.945,Z 852.377,A 0.000,B 0.000,C 90.000,E1 283.772} C_DIS
LIN {X -0.286,Y -663.648,Z 852.374,A 0.000,B 0.000,C 90.000,E1 283.300} C_DIS
LIN {X 0.096,Y -664.281,Z 852.370,A 0.000,B 0.000,C 90.000,E1 282.535} C_DIS
LIN {X -0.078,Y -664.493,Z 852.367,A 0.000,B 0.000,C 90.000,E1 282.063} C_DIS
LIN {X -0.255,Y -664.509,Z 852.364,A 0.000,B 0.000,C 90.000,E1 281.591} C_DIS
LIN {X 0.000,Y -664.074,Z 852.360,A 0.000,B 0.000,C 90.000,E1 280.838} C_DIS
LIN {X -0.182,Y -663.581,Z 852.358,A 0.000,B 0.000,C 90.000,E1 280.366} C_DIS
LIN {X 0.165,Y -662.838,Z 852.355,A 0.000,B 0.000,C 90.000,E1 279.849} C_DIS
LIN {X -0.031,Y -661.734,Z 852.352,A 0.000,B 0.000,C 90.000,E1 279.378} C_DIS
LIN {X 0.309,Y -660.339,Z 852.349,A 0.000,B 0.000,C 90.000,E1 278.859} C_DIS
LIN {X -0.008,Y -658.561,Z 852.347,A 0.000,B 0.000,C 90.000,E1 278.398} C_DIS
LIN {X -0.332,Y -656.484,Z 852.344,A 0.000,B 0.000,C 90.000,E1 277.936} C_DIS
LIN {X 0.090,Y -654.699,Z 852.342,A 0.000,B 0.000,C 90.000,E1 277.530} C_DIS
LIN {X -0.259,Y -651.962,Z 852.339,A 0.000,B 0.000,C 90.000,E1 277.068} C_DIS
LIN {X 0.022,Y -648.909,Z 852.336,A 0.000,B 0.000,C 90.000,E1 276.549} C_DIS
LIN {X 0.281,Y -645.344,Z 852.334,A 0.000,B 0.000,C 90.000,E1 276.030} C_DIS
LIN {X -0.127,Y -641.180,Z 852.331,A 0.000,B 0.000,C 90.000,E1 275.568} C_DIS
LIN {X 0.202,Y -637.475,Z 852.329,A 0.000,B 0.000,C 90.000,E1 275.163} C_DIS
LIN {X 0.057,Y -635.064,Z 852.328,A 0.000,B 0.000,C 90.000,E1 274.935} C_DIS
LIN {X -0.111,Y -632.182,Z 852.326,A 0.000,B 0.000,C 90.000,E1 274.702} C_DIS
LIN {X -0.002,Y -626.349,Z 852.324,A 0.000,B 0.000,C 90.000,E1 274.245} C_DIS
LIN {X 0.244,Y -623.271,Z 852.322,A 0.000,B 0.000,C 90.000,E1 274.012} C_DIS
LIN {X 0.036,Y -617.641,Z 852.320,A 0.000,B 0.000,C 90.000,E1 273.669} C_DIS
LIN {X -0.307,Y -611.208,Z 852.318,A 0.000,B 0.000,C 90.000,E1 273.326} C_DIS
LIN {X 0.081,Y -602.374,Z 852.316,A 0.000,B 0.000,C 90.000,E1 272.865} C_DIS
LIN {X 0.042,Y -597.195,Z 852.315,A 0.000,B 0.000,C 90.000,E1 272.636} C_DIS
LIN {X 0.169,Y -589.801,Z 852.313,A 0.000,B 0.000,C 90.000,E1 272.350} C_DIS
LIN {X 0.174,Y -584.125,Z 852.312,A 0.000,B 0.000,C 90.000,E1 272.178} C_DIS
LIN {X -0.072,Y -578.186,Z 852.311,A 0.000,B 0.000,C 90.000,E1 272.064} C_DIS
LIN {X 0.004,Y -571.261,Z 852.311,A 0.000,B 0.000,C 90.000,E1 271.949} C_DIS
LIN {X -0.012,Y -564.369,Z 852.311,A 0.000,B 0.000,C 90.000,E1 271.892} C_DIS
LIN {X -0.228,Y -557.050,Z 852.310,A 0.000,B 0.000,C 90.000,E1 271.892} C_DIS
LIN {X 0.045,Y -552.866,Z 852.310,A 0.000,B 0.000,C 90.000,E1 271.835} C_DIS
LIN {X 0.126,Y -549.604,Z 852.310,A 0.000,B 0.000,C 90.000,E1 271.718} C_DIS
LIN {X 0.092,Y -549.536,Z 852.310,A 0.000,B 0.000,C 90.000,E1 271.718} C_DIS
LIN {X 0.061,Y -548.273,Z 852.308,A 0.000,B 0.000,C 90.000,E1 271.489} C_DIS
LIN {X -0.261,Y -547.205,Z 852.306,A 0.000,B 0.000,C 90.000,E1 271.088} C_DIS
LIN {X -0.124,Y -546.151,Z 852.301,A 0.000,B 0.000,C 90.000,E1 270.229} C_DIS
LIN {X 0.206,Y -544.329,Z 852.289,A 0.000,B 0.000,C 90.000,E1 267.936} C_DIS
LIN {X -0.123,Y -543.110,Z 852.279,A 0.000,B 0.000,C 90.000,E1 266.274} C_DIS
LIN {X 0.051,Y -542.368,Z 852.273,A 0.000,B 0.000,C 90.000,E1 265.122} C_DIS
LIN {X 0.231,Y -541.335,Z 852.265,A 0.000,B 0.000,C 90.000,E1 263.685} C_DIS
LIN {X -0.160,Y -540.324,Z 852.259,A 0.000,B 0.000,C 90.000,E1 262.591} C_DIS
LIN {X 0.176,Y -538.838,Z 852.249,A 0.000,B 0.000,C 90.000,E1 260.849} C_DIS
LIN {X -0.110,Y -537.446,Z 852.241,A 0.000,B 0.000,C 90.000,E1 259.454} C_DIS
LIN {X 0.142,Y -536.352,Z 852.235,A 0.000,B 0.000,C 90.000,E1 258.285} C_DIS
LIN {X -0.092,Y -534.837,Z 852.227,A 0.000,B 0.000,C 90.000,E1 256.881} C_DIS
LIN {X -0.011,Y -532.382,Z 852.216,A 0.000,B 0.000,C 90.000,E1 254.866} C_DIS
LIN {X -0.024,Y -530.391,Z 852.206,A 0.000,B 0.000,C 90.000,E1 253.142} C_DIS
LIN {X 0.053,Y -528.624,Z 852.198,A 0.000,B 0.000,C 90.000,E1 251.692} C_DIS
LIN {X 0.098,Y -526.787,Z 852.190,A 0.000,B 0.000,C 90.000,E1 250.242} C_DIS
LIN {X -0.228,Y -524.469,Z 852.181,A 0.000,B 0.000,C 90.000,E1 248.539} C_DIS
LIN {X -0.221,Y -521.933,Z 852.171,A 0.000,B 0.000,C 90.000,E1 246.794} C_DIS
LIN {X 0.058,Y -519.710,Z 852.163,A 0.000,B 0.000,C 90.000,E1 245.305} C_DIS
LIN {X 0.231,Y -518.368,Z 852.158,A 0.000,B 0.000,C 90.000,E1 244.409} C_DIS
LIN {X 0.057,Y -516.398,Z 852.151,A 0.000,B 0.000,C 90.000,E1 243.256} C_DIS
LIN {X 0.211,Y -512.797,Z 852.140,A 0.000,B 0.000,C 90.000,E1 241.179} C_DIS
LIN {X 0.198,Y -510.696,Z 852.133,A 0.000,B 0.000,C 90.000,E1 239.999} C_DIS
LIN {X -0.062,Y -507.349,Z 852.124,A 0.000,B 0.000,C 90.000,E1 238.250} C_DIS
LIN {X 0.101,Y -505.045,Z 852.117,A 0.000,B 0.000,C 90.000,E1 237.041} C_DIS
LIN {X -0.199,Y -502.528,Z 852.110,A 0.000,B 0.000,C 90.000,E1 235.881} C_DIS
LIN {X -0.255,Y -499.868,Z 852.104,A 0.000,B 0.000,C 90.000,E1 234.689} C_DIS
LIN {X -0.221,Y -497.700,Z 852.099,A 0.000,B 0.000,C 90.000,E1 233.783} C_DIS
LIN {X 0.213,Y -492.772,Z 852.087,A 0.000,B 0.000,C 90.000,E1 231.618} C_DIS
LIN {X -0.088,Y -488.447,Z 852.077,A 0.000,B 0.000,C 90.000,E1 229.828} C_DIS
LIN {X 0.018,Y -484.976,Z 852.068,A 0.000,B 0.000,C 90.000,E1 228.286} C_DIS
LIN {X -0.011,Y -480.162,Z 852.056,A 0.000,B 0.000,C 90.000,E1 226.134} C_DIS
LIN {X 0.032,Y -476.272,Z 852.046,A 0.000,B 0.000,C 90.000,E1 224.271} C_DIS
LIN {X 0.183,Y -470.865,Z 852.032,A 0.000,B 0.000,C 90.000,E1 221.757} C_DIS
LIN {X 0.071,Y -466.796,Z 852.022,A 0.000,B 0.000,C 90.000,E1 219.886} C_DIS
LIN {X 0.114,Y -463.481,Z 852.013,A 0.000,B 0.000,C 90.000,E1 218.302} C_DIS
LIN {X -0.117,Y -460.186,Z 852.004,A 0.000,B 0.000,C 90.000,E1 216.744} C_DIS
LIN {X 0.014,Y -458.906,Z 852.001,A 0.000,B 0.000,C 90.000,E1 216.091} C_DIS
LIN {X -0.197,Y -454.760,Z 851.990,A 0.000,B 0.000,C 90.000,E1 214.199} C_DIS
LIN {X 0.034,Y -449.245,Z 851.976,A 0.000,B 0.000,C 90.000,E1 211.592} C_DIS
LIN {X -0.008,Y -443.777,Z 851.961,A 0.000,B 0.000,C 90.000,E1 208.999} C_DIS
LIN {X -0.170,Y -440.434,Z 851.952,A 0.000,B 0.000,C 90.000,E1 207.385} C_DIS
LIN {X -0.003,Y -437.074,Z 851.943,A 0.000,B 0.000,C 90.000,E1 205.720} C_DIS
LIN {X -0.093,Y -433.715,Z 851.934,A 0.000,B 0.000,C 90.000,E1 204.079} C_DIS
LIN {X -0.044,Y -429.657,Z 851.923,A 0.000,B 0.000,C 90.000,E1 202.078} C_DIS
LIN {X -0.210,Y -426.420,Z 851.913,A 0.000,B 0.000,C 90.000,E1 200.429} C_DIS
LIN {X -0.068,Y -421.843,Z 851.900,A 0.000,B 0.000,C 90.000,E1 198.055} C_DIS
LIN {X -0.128,Y -418.625,Z 851.891,A 0.000,B 0.000,C 90.000,E1 196.370} C_DIS
LIN {X -0.122,Y -415.812,Z 851.883,A 0.000,B 0.000,C 90.000,E1 195.009} C_DIS
LIN {X -0.156,Y -412.992,Z 851.876,A 0.000,B 0.000,C 90.000,E1 193.647} C_DIS
LIN {X -0.146,Y -407.655,Z 851.860,A 0.000,B 0.000,C 90.000,E1 190.894} C_DIS
LIN {X -0.069,Y -404.290,Z 851.851,A 0.000,B 0.000,C 90.000,E1 189.151} C_DIS
LIN {X -0.065,Y -400.825,Z 851.841,A 0.000,B 0.000,C 90.000,E1 187.409} C_DIS
LIN {X -0.145,Y -393.949,Z 851.820,A 0.000,B 0.000,C 90.000,E1 183.555} C_DIS
LIN {X 0.055,Y -389.764,Z 851.804,A 0.000,B 0.000,C 90.000,E1 180.688} C_DIS
LIN {X -0.093,Y -386.889,Z 851.792,A 0.000,B 0.000,C 90.000,E1 178.568} C_DIS
LIN {X -0.018,Y -383.383,Z 851.778,A 0.000,B 0.000,C 90.000,E1 176.045} C_DIS
LIN {X -0.145,Y -380.971,Z 851.768,A 0.000,B 0.000,C 90.000,E1 174.261} C_DIS
LIN {X 0.007,Y -378.310,Z 851.756,A 0.000,B 0.000,C 90.000,E1 172.064} C_DIS
LIN {X -0.174,Y -374.827,Z 851.738,A 0.000,B 0.000,C 90.000,E1 168.814} C_DIS
LIN {X 0.144,Y -372.308,Z 851.717,A 0.000,B 0.000,C 90.000,E1 165.102} C_DIS
LIN {X 0.091,Y -371.999,Z 851.705,A 0.000,B 0.000,C 90.000,E1 162.906} C_DIS
LIN {X 0.057,Y -372.023,Z 851.703,A 0.000,B 0.000,C 90.000,E1 162.543} C_DIS
LIN {X -0.072,Y -373.125,Z 851.695,A 0.000,B 0.000,C 90.000,E1 161.094} C_DIS
LIN {X -0.131,Y -374.151,Z 851.691,A 0.000,B 0.000,C 90.000,E1 160.369} C_DIS
LIN {X -0.056,Y -375.487,Z 851.687,A 0.000,B 0.000,C 90.000,E1 159.625} C_DIS
LIN {X -0.068,Y -375.992,Z 851.686,A 0.000,B 0.000,C 90.000,E1 159.444} C_DIS
LIN {X -0.099,Y -377.964,Z 851.683,A 0.000,B 0.000,C 90.000,E1 158.901} C_DIS
LIN {X -0.113,Y -379.130,Z 851.681,A 0.000,B 0.000,C 90.000,E1 158.539} C_DIS
LIN {X 0.014,Y -380.737,Z 851.679,A 0.000,B 0.000,C 90.000,E1 158.156} C_DIS
LIN {X -0.174,Y -385.748,Z 851.675,A 0.000,B 0.000,C 90.000,E1 157.486} C_DIS
LIN {X -0.024,Y -387.329,Z 851.674,A 0.000,B 0.000,C 90.000,E1 157.283} C_DIS
LIN {X -0.095,Y -393.115,Z 851.671,A 0.000,B 0.000,C 90.000,E1 156.869} C_DIS
LIN {X 0.003,Y -407.981,Z 851.668,A 0.000,B 0.000,C 90.000,E1 156.230} C_DIS
LIN {X -0.108,Y -411.678,Z 851.667,A 0.000,B 0.000,C 90.000,E1 156.102} C_DIS
LIN {X 0.125,Y -422.050,Z 851.665,A 0.000,B 0.000,C 90.000,E1 155.613} C_DIS
LIN {X -0.081,Y -425.422,Z 851.664,A 0.000,B 0.000,C 90.000,E1 155.485} C_DIS
LIN {X -0.005,Y -434.785,Z 851.661,A 0.000,B 0.000,C 90.000,E1 154.921} C_DIS
LIN {X -0.003,Y -444.266,Z 851.657,A 0.000,B 0.000,C 90.000,E1 154.280} C_DIS
LIN {X 0.016,Y -450.489,Z 851.655,A 0.000,B 0.000,C 90.000,E1 153.819} C_DIS
LIN {X -0.016,Y -455.154,Z 851.653,A 0.000,B 0.000,C 90.000,E1 153.461} C_DIS
LIN {X -0.021,Y -462.487,Z 851.649,A 0.000,B 0.000,C 90.000,E1 152.820} C_DIS
LIN {X -0.054,Y -466.737,Z 851.647,A 0.000,B 0.000,C 90.000,E1 152.410} C_DIS
LIN {X -0.137,Y -473.516,Z 851.643,A 0.000,B 0.000,C 90.000,E1 151.691} C_DIS
LIN {X 0.101,Y -480.401,Z 851.639,A 0.000,B 0.000,C 90.000,E1 150.923} C_DIS
LIN {X -0.180,Y -490.698,Z 851.632,A 0.000,B 0.000,C 90.000,E1 149.744} C_DIS
LIN {X 0.058,Y -495.454,Z 851.629,A 0.000,B 0.000,C 90.000,E1 149.125} C_DIS
LIN {X 0.261,Y -499.081,Z 851.626,A 0.000,B 0.000,C 90.000,E1 148.663} C_DIS
LIN {X 0.164,Y -503.396,Z 851.623,A 0.000,B 0.000,C 90.000,E1 148.074} C_DIS
LIN {X -0.153,Y -506.797,Z 851.620,A 0.000,B 0.000,C 90.000,E1 147.661} C_DIS
LIN {X -0.218,Y -513.914,Z 851.615,A 0.000,B 0.000,C 90.000,E1 146.628} C_DIS
LIN {X -0.190,Y -520.257,Z 851.609,A 0.000,B 0.000,C 90.000,E1 145.595} C_DIS
LIN {X 0.050,Y -526.990,Z 851.602,A 0.000,B 0.000,C 90.000,E1 144.402} C_DIS
LIN {X -0.172,Y -531.022,Z 851.598,A 0.000,B 0.000,C 90.000,E1 143.703} C_DIS
LIN {X -0.013,Y -541.207,Z 851.588,A 0.000,B 0.000,C 90.000,E1 141.823} C_DIS
LIN {X -0.087,Y -549.960,Z 851.579,A 0.000,B 0.000,C 90.000,E1 140.275} C_DIS
LIN {X -0.347,Y -554.572,Z 851.575,A 0.000,B 0.000,C 90.000,E1 139.461} C_DIS
LIN {X -0.227,Y -562.578,Z 851.566,A 0.000,B 0.000,C 90.000,E1 137.919} C_DIS
LIN {X -0.128,Y -567.832,Z 851.561,A 0.000,B 0.000,C 90.000,E1 136.944} C_DIS
LIN {X -0.322,Y -575.923,Z 851.552,A 0.000,B 0.000,C 90.000,E1 135.324} C_DIS
LIN {X -0.080,Y -580.467,Z 851.546,A 0.000,B 0.000,C 90.000,E1 134.352} C_DIS
LIN {X -0.064,Y -584.432,Z 851.542,A 0.000,B 0.000,C 90.000,E1 133.542} C_DIS
LIN {X 0.064,Y -590.143,Z 851.535,A 0.000,B 0.000,C 90.000,E1 132.324} C_DIS
LIN {X 0.141,Y -595.985,Z 851.528,A 0.000,B 0.000,C 90.000,E1 130.987} C_DIS
LIN {X 0.372,Y -601.526,Z 851.521,A 0.000,B 0.000,C 90.000,E1 129.644} C_DIS
LIN {X -0.199,Y -604.665,Z 851.516,A 0.000,B 0.000,C 90.000,E1 128.910} C_DIS
LIN {X -0.098,Y -608.511,Z 851.510,A 0.000,B 0.000,C 90.000,E1 127.855} C_DIS
LIN {X 0.080,Y -612.727,Z 851.503,A 0.000,B 0.000,C 90.000,E1 126.537} C_DIS
LIN {X 0.161,Y -617.486,Z 851.494,A 0.000,B 0.000,C 90.000,E1 124.978} C_DIS
LIN {X -0.315,Y -619.946,Z 851.489,A 0.000,B 0.000,C 90.000,E1 123.992} C_DIS
LIN {X 0.292,Y -621.633,Z 851.484,A 0.000,B 0.000,C 90.000,E1 123.166} C_DIS
LIN {X -0.158,Y -624.070,Z 851.477,A 0.000,B 0.000,C 90.000,E1 121.926} C_DIS
LIN {X 0.160,Y -625.445,Z 851.473,A 0.000,B 0.000,C 90.000,E1 121.131} C_DIS
LIN {X -0.010,Y -627.723,Z 851.465,A 0.000,B 0.000,C 90.000,E1 119.617} C_DIS
LIN {X -0.200,Y -628.629,Z 851.460,A 0.000,B 0.000,C 90.000,E1 118.871} C_DIS
LIN {X -0.135,Y -629.339,Z 851.456,A 0.000,B 0.000,C 90.000,E1 118.103} C_DIS
LIN {X -0.030,Y -629.987,Z 851.450,A 0.000,B 0.000,C 90.000,E1 117.078} C_DIS
LIN {X 0.057,Y -630.131,Z 851.446,A 0.000,B 0.000,C 90.000,E1 116.309} C_DIS
LIN {X 0.116,Y -630.101,Z 851.443,A 0.000,B 0.000,C 90.000,E1 115.796} C_DIS
LIN {X 0.145,Y -629.992,Z 851.442,A 0.000,B 0.000,C 90.000,E1 115.540} C_DIS
LIN {X 0.252,Y -629.205,Z 851.436,A 0.000,B 0.000,C 90.000,E1 114.515} C_DIS
LIN {X 0.063,Y -627.937,Z 851.432,A 0.000,B 0.000,C 90.000,E1 113.770} C_DIS
LIN {X 0.097,Y -626.641,Z 851.429,A 0.000,B 0.000,C 90.000,E1 113.259} C_DIS
LIN {X -0.123,Y -624.363,Z 851.427,A 0.000,B 0.000,C 90.000,E1 112.770} C_DIS
LIN {X -0.117,Y -622.784,Z 851.425,A 0.000,B 0.000,C 90.000,E1 112.514} C_DIS
LIN {X -0.118,Y -620.788,Z 851.424,A 0.000,B 0.000,C 90.000,E1 112.259} C_DIS
LIN {X -0.356,Y -619.622,Z 851.423,A 0.000,B 0.000,C 90.000,E1 112.153} C_DIS
LIN {X -0.043,Y -613.616,Z 851.420,A 0.000,B 0.000,C 90.000,E1 111.589} C_DIS
LIN {X 0.196,Y -608.962,Z 851.418,A 0.000,B 0.000,C 90.000,E1 111.227} C_DIS
LIN {X 0.203,Y -600.951,Z 851.415,A 0.000,B 0.000,C 90.000,E1 110.737} C_DIS
LIN {X 0.202,Y -594.422,Z 851.413,A 0.000,B 0.000,C 90.000,E1 110.375} C_DIS
LIN {X -0.178,Y -585.846,Z 851.411,A 0.000,B 0.000,C 90.000,E1 109.993} C_DIS
LIN {X 0.027,Y -576.834,Z 851.409,A 0.000,B 0.000,C 90.000,E1 109.631} C_DIS
LIN {X -0.186,Y -569.705,Z 851.408,A 0.000,B 0.000,C 90.000,E1 109.396} C_DIS
LIN {X -0.106,Y -568.108,Z 851.407,A 0.000,B 0.000,C 90.000,E1 109.322} C_DIS
LIN {X -0.215,Y -567.028,Z 851.407,A 0.000,B 0.000,C 90.000,E1 109.268} C_DIS
LIN {X 0.279,Y -564.197,Z 851.406,A 0.000,B 0.000,C 90.000,E1 108.960} C_DIS
LIN {X 0.144,Y -562.944,Z 851.404,A 0.000,B 0.000,C 90.000,E1 108.779} C_DIS
LIN {X 0.102,Y -561.368,Z 851.401,A 0.000,B 0.000,C 90.000,E1 108.236} C_DIS
LIN {X -0.137,Y -560.829,Z 851.400,A 0.000,B 0.000,C 90.000,E1 107.928} C_DIS
LIN {X 0.133,Y -560.469,Z 851.396,A 0.000,B 0.000,C 90.000,E1 107.347} C_DIS
LIN {X -0.170,Y -560.376,Z 851.387,A 0.000,B 0.000,C 90.000,E1 105.717} C_DIS
LIN {X -0.060,Y -561.375,Z 851.372,A 0.000,B 0.000,C 90.000,E1 102.939} C_DIS
LIN {X -0.083,Y -562.551,Z 851.361,A 0.000,B 0.000,C 90.000,E1 101.007} C_DIS
LIN {X 0.212,Y -563.718,Z 851.352,A 0.000,B 0.000,C 90.000,E1 99.321} C_DIS
LIN {X -0.109,Y -564.898,Z 851.343,A 0.000,B 0.000,C 90.000,E1 97.701} C_DIS
LIN {X -0.009,Y -565.677,Z 851.335,A 0.000,B 0.000,C 90.000,E1 96.315} C_DIS
LIN {X -0.059,Y -566.231,Z 851.329,A 0.000,B 0.000,C 90.000,E1 95.220} C_DIS
LIN {X 0.004,Y -566.871,Z 851.321,A 0.000,B 0.000,C 90.000,E1 93.841} C_DIS
LIN {X 0.041,Y -567.331,Z 851.314,A 0.000,B 0.000,C 90.000,E1 92.465} C_DIS
LIN {X 0.088,Y -567.698,Z 851.306,A 0.000,B 0.000,C 90.000,E1 91.088} C_DIS
LIN {X 0.129,Y -568.060,Z 851.299,A 0.000,B 0.000,C 90.000,E1 89.714} C_DIS
LIN {X -0.131,Y -568.501,Z 851.288,A 0.000,B 0.000,C 90.000,E1 87.822} C_DIS
LIN {X -0.060,Y -568.725,Z 851.280,A 0.000,B 0.000,C 90.000,E1 86.445} C_DIS
LIN {X -0.236,Y -569.051,Z 851.270,A 0.000,B 0.000,C 90.000,E1 84.546} C_DIS
LIN {X 0.157,Y -569.440,Z 851.259,A 0.000,B 0.000,C 90.000,E1 82.591} C_DIS
LIN {X 0.129,Y -569.954,Z 851.248,A 0.000,B 0.000,C 90.000,E1 80.679} C_DIS
LIN {X 0.023,Y -570.509,Z 851.239,A 0.000,B 0.000,C 90.000,E1 79.050} C_DIS
LIN {X -0.150,Y -571.063,Z 851.232,A 0.000,B 0.000,C 90.000,E1 77.701} C_DIS
LIN {X 0.012,Y -571.608,Z 851.223,A 0.000,B 0.000,C 90.000,E1 76.047} C_DIS
LIN {X -0.001,Y -571.898,Z 851.215,A 0.000,B 0.000,C 90.000,E1 74.685} C_DIS
LIN {X 0.164,Y -572.213,Z 851.206,A 0.000,B 0.000,C 90.000,E1 73.032} C_DIS
LIN {X 0.109,Y -572.351,Z 851.197,A 0.000,B 0.000,C 90.000,E1 71.402} C_DIS
LIN {X -0.127,Y -572.217,Z 851.186,A 0.000,B 0.000,C 90.000,E1 69.518} C_DIS
LIN {X -0.169,Y -572.111,Z 851.176,A 0.000,B 0.000,C 90.000,E1 67.614} C_DIS
LIN {X -0.127,Y -571.926,Z 851.167,A 0.000,B 0.000,C 90.000,E1 65.973} C_DIS
LIN {X 0.087,Y -571.573,Z 851.159,A 0.000,B 0.000,C 90.000,E1 64.588} C_DIS
LIN {X 0.115,Y -570.987,Z 851.150,A 0.000,B 0.000,C 90.000,E1 62.948} C_DIS
LIN {X 0.210,Y -570.645,Z 851.144,A 0.000,B 0.000,C 90.000,E1 61.847} C_DIS
LIN {X -0.093,Y -569.933,Z 851.136,A 0.000,B 0.000,C 90.000,E1 60.511} C_DIS
LIN {X 0.162,Y -569.414,Z 851.132,A 0.000,B 0.000,C 90.000,E1 59.665} C_DIS
LIN {X 0.029,Y -568.422,Z 851.126,A 0.000,B 0.000,C 90.000,E1 58.584} C_DIS
LIN {X -0.113,Y -567.371,Z 851.119,A 0.000,B 0.000,C 90.000,E1 57.502} C_DIS
LIN {X -0.272,Y -566.030,Z 851.113,A 0.000,B 0.000,C 90.000,E1 56.421} C_DIS
LIN {X -0.141,Y -564.498,Z 851.107,A 0.000,B 0.000,C 90.000,E1 55.308} C_DIS
LIN {X -0.139,Y -563.213,Z 851.103,A 0.000,B 0.000,C 90.000,E1 54.482} C_DIS
LIN {X 0.176,Y -561.805,Z 851.098,A 0.000,B 0.000,C 90.000,E1 53.623} C_DIS
LIN {X -0.310,Y -560.221,Z 851.093,A 0.000,B 0.000,C 90.000,E1 52.844} C_DIS
LIN {X -0.030,Y -558.436,Z 851.089,A 0.000,B 0.000,C 90.000,E1 51.984} C_DIS
LIN {X -0.209,Y -556.406,Z 851.084,A 0.000,B 0.000,C 90.000,E1 51.170} C_DIS
LIN {X 0.020,Y -554.101,Z 851.080,A 0.000,B 0.000,C 90.000,E1 50.312} C_DIS
LIN {X 0.087,Y -552.443,Z 851.076,A 0.000,B 0.000,C 90.000,E1 49.747} C_DIS
LIN {X -0.153,Y -549.617,Z 851.072,A 0.000,B 0.000,C 90.000,E1 48.933} C_DIS
LIN {X -0.063,Y -546.358,Z 851.067,A 0.000,B 0.000,C 90.000,E1 48.081} C_DIS
LIN {X -0.204,Y -543.473,Z 851.063,A 0.000,B 0.000,C 90.000,E1 47.391} C_DIS
LIN {X 0.200,Y -540.947,Z 851.060,A 0.000,B 0.000,C 90.000,E1 46.782} C_DIS
LIN {X -0.013,Y -537.421,Z 851.056,A 0.000,B 0.000,C 90.000,E1 46.095} C_DIS
LIN {X -0.037,Y -534.378,Z 851.053,A 0.000,B 0.000,C 90.000,E1 45.526} C_DIS
LIN {X 0.282,Y -531.026,Z 851.050,A 0.000,B 0.000,C 90.000,E1 44.919} C_DIS
LIN {X 0.201,Y -527.439,Z 851.047,A 0.000,B 0.000,C 90.000,E1 44.352} C_DIS
LIN {X 0.095,Y -523.570,Z 851.043,A 0.000,B 0.000,C 90.000,E1 43.785} C_DIS
LIN {X 0.103,Y -518.178,Z 851.039,A 0.000,B 0.000,C 90.000,E1 43.056} C_DIS
LIN {X 0.172,Y -514.788,Z 851.037,A 0.000,B 0.000,C 90.000,E1 42.609} C_DIS
LIN {X -0.029,Y -509.918,Z 851.034,A 0.000,B 0.000,C 90.000,E1 42.043} C_DIS
LIN {X 0.047,Y -502.191,Z 851.029,A 0.000,B 0.000,C 90.000,E1 41.148} C_DIS
LIN {X -0.193,Y -495.212,Z 851.025,A 0.000,B 0.000,C 90.000,E1 40.458} C_DIS
LIN {X 0.054,Y -490.921,Z 851.022,A 0.000,B 0.000,C 90.000,E1 40.011} C_DIS
LIN {X -0.174,Y -486.688,Z 851.020,A 0.000,B 0.000,C 90.000,E1 39.644} C_DIS
LIN {X -0.123,Y -479.289,Z 851.017,A 0.000,B 0.000,C 90.000,E1 38.991} C_DIS
LIN {X 0.060,Y -471.712,Z 851.013,A 0.000,B 0.000,C 90.000,E1 38.338} C_DIS
LIN {X 0.029,Y -459.245,Z 851.008,A 0.000,B 0.000,C 90.000,E1 37.363} C_DIS
LIN {X -0.167,Y -449.717,Z 851.004,A 0.000,B 0.000,C 90.000,E1 36.664} C_DIS
LIN {X -0.009,Y -437.158,Z 850.998,A 0.000,B 0.000,C 90.000,E1 35.678} C_DIS
LIN {X 0.080,Y -417.164,Z 850.989,A 0.000,B 0.000,C 90.000,E1 34.040} C_DIS
LIN {X -0.047,Y -403.722,Z 850.982,A 0.000,B 0.000,C 90.000,E1 32.832} C_DIS
LIN {X -0.053,Y -398.250,Z 850.979,A 0.000,B 0.000,C 90.000,E1 32.212} C_DIS
LIN {X -0.040,Y -395.666,Z 850.977,A 0.000,B 0.000,C 90.000,E1 31.878} C_DIS
LIN {X -0.198,Y -393.137,Z 850.975,A 0.000,B 0.000,C 90.000,E1 31.465} C_DIS
LIN {X 0.035,Y -392.274,Z 850.973,A 0.000,B 0.000,C 90.000,E1 31.052} C_DIS
LIN {X -0.058,Y -390.374,Z 850.967,A 0.000,B 0.000,C 90.000,E1 30.001} C_DIS
LIN {X 0.077,Y -390.254,Z 850.962,A 0.000,B 0.000,C 90.000,E1 29.077} C_DIS
LIN {X 0.134,Y -392.514,Z 850.940,A 0.000,B 0.000,C 90.000,E1 25.155} C_DIS
LIN {X 0.042,Y -394.785,Z 850.924,A 0.000,B 0.000,C 90.000,E1 22.333} C_DIS
LIN {X -0.121,Y -397.054,Z 850.910,A 0.000,B 0.000,C 90.000,E1 19.885} C_DIS
LIN {X 0.107,Y -400.069,Z 850.895,A 0.000,B 0.000,C 90.000,E1 17.040} C_DIS
LIN {X 0.084,Y -403.603,Z 850.879,A 0.000,B 0.000,C 90.000,E1 14.245} C_DIS
LIN {X -0.031,Y -407.144,Z 850.866,A 0.000,B 0.000,C 90.000,E1 11.827} C_DIS
LIN {X 0.152,Y -410.461,Z 850.854,A 0.000,B 0.000,C 90.000,E1 9.726} C_DIS
LIN {X -0.086,Y -414.537,Z 850.841,A 0.000,B 0.000,C 90.000,E1 7.352} C_DIS
LIN {X 0.110,Y -418.804,Z 850.828,A 0.000,B 0.000,C 90.000,E1 4.935} C_DIS
LIN {X 0.129,Y -425.547,Z 850.809,A 0.000,B 0.000,C 90.000,E1 1.547} C_DIS
LIN {X -0.197,Y -430.251,Z 850.797,A 0.000,B 0.000,C 90.000,E1 359.484} C_DIS
LIN {X -0.050,Y -435.867,Z 850.784,A 0.000,B 0.000,C 90.000,E1 357.135} C_DIS
LIN {X 0.054,Y -439.974,Z 850.775,A 0.000,B 0.000,C 90.000,E1 355.469} C_DIS
LIN {X -0.045,Y -445.314,Z 850.764,A 0.000,B 0.000,C 90.000,E1 353.514} C_DIS
LIN {X 0.183,Y -447.010,Z 850.761,A 0.000,B 0.000,C 90.000,E1 352.996} C_DIS
LIN {X -0.147,Y -447.668,Z 850.760,A 0.000,B 0.000,C 90.000,E1 352.875} C_DIS
LIN {X -0.023,Y -449.542,Z 850.759,A 0.000,B 0.000,C 90.000,E1 352.534} C_DIS
LIN {X -0.090,Y -450.868,Z 850.757,A 0.000,B 0.000,C 90.000,E1 352.299} C_DIS
LIN {X 0.010,Y -452.730,Z 850.756,A 0.000,B 0.000,C 90.000,E1 352.064} C_DIS
LIN {X 0.107,Y -454.383,Z 850.755,A 0.000,B 0.000,C 90.000,E1 351.894} C_DIS
LIN {X -0.073,Y -457.821,Z 850.754,A 0.000,B 0.000,C 90.000,E1 351.659} C_DIS
LIN {X -0.138,Y -465.160,Z 850.751,A 0.000,B 0.000,C 90.000,E1 351.254} C_DIS
LIN {X 0.049,Y -474.908,Z 850.749,A 0.000,B 0.000,C 90.000,E1 350.735} C_DIS
LIN {X 0.001,Y -481.597,Z 850.747,A 0.000,B 0.000,C 90.000,E1 350.387} C_DIS
LIN {X 0.215,Y -491.239,Z 850.744,A 0.000,B 0.000,C 90.000,E1 349.803} C_DIS
LIN {X -0.145,Y -503.798,Z 850.739,A 0.000,B 0.000,C 90.000,E1 349.050} C_DIS
LIN {X -0.005,Y -513.289,Z 850.736,A 0.000,B 0.000,C 90.000,E1 348.409} C_DIS
LIN {X 0.074,Y -522.478,Z 850.732,A 0.000,B 0.000,C 90.000,E1 347.757} C_DIS
LIN {X -0.213,Y -531.552,Z 850.728,A 0.000,B 0.000,C 90.000,E1 347.117} C_DIS
LIN {X -0.136,Y -543.199,Z 850.723,A 0.000,B 0.000,C 90.000,E1 346.172} C_DIS
LIN {X -0.270,Y -548.763,Z 850.720,A 0.000,B 0.000,C 90.000,E1 345.700} C_DIS
LIN {X 0.000,Y -554.263,Z 850.718,A 0.000,B 0.000,C 90.000,E1 345.172} C_DIS
LIN {X 0.029,Y -562.203,Z 850.713,A 0.000,B 0.000,C 90.000,E1 344.393} C_DIS
LIN {X -0.055,Y -567.175,Z 850.710,A 0.000,B 0.000,C 90.000,E1 343.866} C_DIS
LIN {X -0.034,Y -575.633,Z 850.705,A 0.000,B 0.000,C 90.000,E1 342.906} C_DIS
LIN {X 0.009,Y -584.169,Z 850.699,A 0.000,B 0.000,C 90.000,E1 341.819} C_DIS
LIN {X 0.007,Y -589.010,Z 850.695,A 0.000,B 0.000,C 90.000,E1 341.148} C_DIS
LIN {X -0.146,Y -593.493,Z 850.692,A 0.000,B 0.000,C 90.000,E1 340.496} C_DIS
LIN {X -0.071,Y -597.667,Z 850.688,A 0.000,B 0.000,C 90.000,E1 339.826} C_DIS
LIN {X 0.000,Y -602.520,Z 850.684,A 0.000,B 0.000,C 90.000,E1 339.028} C_DIS
LIN {X 0.034,Y -609.274,Z 850.677,A 0.000,B 0.000,C 90.000,E1 337.847} C_DIS
LIN {X 0.192,Y -614.947,Z 850.671,A 0.000,B 0.000,C 90.000,E1 336.794} C_DIS
LIN {X -0.127,Y -618.963,Z 850.667,A 0.000,B 0.000,C 90.000,E1 336.049} C_DIS
LIN {X -0.155,Y -622.834,Z 850.663,A 0.000,B 0.000,C 90.000,E1 335.281} C_DIS
LIN {X 0.178,Y -628.236,Z 850.656,A 0.000,B 0.000,C 90.000,E1 334.101} C_DIS
LIN {X -0.323,Y -631.652,Z 850.652,A 0.000,B 0.000,C 90.000,E1 333.384} C_DIS
LIN {X -0.141,Y -636.778,Z 850.645,A 0.000,B 0.000,C 90.000,E1 332.103} C_DIS
LIN {X 0.368,Y -640.712,Z 850.639,A 0.000,B 0.000,C 90.000,E1 331.051} C_DIS
LIN {X 0.059,Y -644.535,Z 850.634,A 0.000,B 0.000,C 90.000,E1 330.078} C_DIS
LIN {X 0.117,Y -648.003,Z 850.628,A 0.000,B 0.000,C 90.000,E1 329.076} C_DIS
LIN {X 0.222,Y -651.337,Z 850.623,A 0.000,B 0.000,C 90.000,E1 328.074} C_DIS
LIN {X -0.194,Y -655.749,Z 850.615,A 0.000,B 0.000,C 90.000,E1 326.628} C_DIS
LIN {X -0.078,Y -659.085,Z 850.608,A 0.000,B 0.000,C 90.000,E1 325.388} C_DIS
LIN {X 0.046,Y -660.865,Z 850.604,A 0.000,B 0.000,C 90.000,E1 324.642} C_DIS
LIN {X -0.408,Y -663.062,Z 850.598,A 0.000,B 0.000,C 90.000,E1 323.703} C_DIS
LIN {X -0.330,Y -665.542,Z 850.591,A 0.000,B 0.000,C 90.000,E1 322.477} C_DIS
LIN {X -0.213,Y -667.525,Z 850.585,A 0.000,B 0.000,C 90.000,E1 321.251} C_DIS
LIN {X -0.151,Y -668.701,Z 850.581,A 0.000,B 0.000,C 90.000,E1 320.517} C_DIS
LIN {X -0.075,Y -670.532,Z 850.573,A 0.000,B 0.000,C 90.000,E1 319.057} C_DIS
LIN {X 0.141,Y -673.366,Z 850.560,A 0.000,B 0.000,C 90.000,E1 316.863} C_DIS
LIN {X 0.230,Y -674.576,Z 850.555,A 0.000,B 0.000,C 90.000,E1 315.891} C_DIS
LIN {X 0.256,Y -674.796,Z 850.554,A 0.000,B 0.000,C 90.000,E1 315.648} C_DIS
LIN {X 0.283,Y -675.203,Z 850.552,A 0.000,B 0.000,C 90.000,E1 315.405} C_DIS
LIN {X 0.098,Y -677.400,Z 850.540,A 0.000,B 0.000,C 90.000,E1 313.257} C_DIS
LIN {X -0.113,Y -679.110,Z 850.531,A 0.000,B 0.000,C 90.000,E1 311.595} C_DIS
LIN {X 0.128,Y -680.237,Z 850.524,A 0.000,B 0.000,C 90.000,E1 310.378} C_DIS
LIN {X 0.116,Y -681.730,Z 850.515,A 0.000,B 0.000,C 90.000,E1 308.705} C_DIS
LIN {X -0.034,Y -682.760,Z 850.508,A 0.000,B 0.000,C 90.000,E1 307.523} C_DIS
LIN {X -0.015,Y -683.939,Z 850.501,A 0.000,B 0.000,C 90.000,E1 306.091} C_DIS
LIN {X -0.181,Y -684.636,Z 850.495,A 0.000,B 0.000,C 90.000,E1 305.152} C_DIS
LIN {X 0.028,Y -685.622,Z 850.487,A 0.000,B 0.000,C 90.000,E1 303.706} C_DIS
LIN {X -0.117,Y -686.804,Z 850.478,A 0.000,B 0.000,C 90.000,E1 302.054} C_DIS
LIN {X -0.174,Y -688.401,Z 850.466,A 0.000,B 0.000,C 90.000,E1 299.922} C_DIS
LIN {X -0.155,Y -690.018,Z 850.456,A 0.000,B 0.000,C 90.000,E1 298.025} C_DIS
LIN {X -0.181,Y -691.971,Z 850.444,A 0.000,B 0.000,C 90.000,E1 295.899} C_DIS
LIN {X -0.185,Y -693.073,Z 850.437,A 0.000,B 0.000,C 90.000,E1 294.719} C_DIS
LIN {X -0.083,Y -693.539,Z 850.433,A 0.000,B 0.000,C 90.000,E1 294.003} C_DIS
LIN {X -0.120,Y -693.603,Z 850.432,A 0.000,B 0.000,C 90.000,E1 293.770} C_DIS
LIN {X 0.367,Y -693.468,Z 850.429,A 0.000,B 0.000,C 90.000,E1 293.259} C_DIS
LIN {X -0.300,Y -693.028,Z 850.428,A 0.000,B 0.000,C 90.000,E1 293.078} C_DIS
LIN {X -0.086,Y -691.380,Z 850.425,A 0.000,B 0.000,C 90.000,E1 292.589} C_DIS
LIN {X 0.032,Y -690.820,Z 850.425,A 0.000,B 0.000,C 90.000,E1 292.461} C_DIS
LIN {X 0.150,Y -689.960,Z 850.424,A 0.000,B 0.000,C 90.000,E1 292.333} C_DIS
LIN {X 0.119,Y -687.664,Z 850.423,A 0.000,B 0.000,C 90.000,E1 292.099} C_DIS
LIN {X -0.287,Y -685.034,Z 850.422,A 0.000,B 0.000,C 90.000,E1 291.897} C_DIS
LIN {X -0.101,Y -683.516,Z 850.421,A 0.000,B 0.000,C 90.000,E1 291.770} C_DIS
LIN {X -0.168,Y -681.109,Z 850.420,A 0.000,B 0.000,C 90.000,E1 291.663} C_DIS
LIN {X -0.290,Y -673.751,Z 850.419,A 0.000,B 0.000,C 90.000,E1 291.408} C_DIS
LIN {X -0.207,Y -669.685,Z 850.418,A 0.000,B 0.000,C 90.000,E1 291.280} C_DIS
LIN {X -0.175,Y -661.500,Z 850.417,A 0.000,B 0.000,C 90.000,E1 291.099} C_DIS
LIN {X -0.143,Y -657.815,Z 850.417,A 0.000,B 0.000,C 90.000,E1 291.025} C_DIS
LIN {X 0.001,Y -649.002,Z 850.416,A 0.000,B 0.000,C 90.000,E1 290.791} C_DIS
LIN {X 0.156,Y -646.197,Z 850.415,A 0.000,B 0.000,C 90.000,E1 290.684} C_DIS
LIN {X -0.071,Y -640.139,Z 850.414,A 0.000,B 0.000,C 90.000,E1 290.429} C_DIS
LIN {X -0.103,Y -637.793,Z 850.412,A 0.000,B 0.000,C 90.000,E1 290.248} C_DIS
LIN {X -0.142,Y -637.767,Z 850.412,A 0.000,B 0.000,C 90.000,E1 290.248} C_DIS
LIN {X -0.254,Y -637.464,Z 850.412,A 0.000,B 0.000,C 90.000,E1 290.120} C_DIS
LIN {X -0.216,Y -638.776,Z 850.409,A 0.000,B 0.000,C 90.000,E1 289.685} C_DIS
LIN {X -0.089,Y -644.099,Z 850.404,A 0.000,B 0.000,C 90.000,E1 288.671} C_DIS
LIN {X -0.224,Y -646.146,Z 850.402,A 0.000,B 0.000,C 90.000,E1 288.308} C_DIS
LIN {X 0.155,Y -649.737,Z 850.398,A 0.000,B 0.000,C 90.000,E1 287.528} C_DIS
LIN {X 0.076,Y -651.946,Z 850.395,A 0.000,B 0.000,C 90.000,E1 287.040} C_DIS
LIN {X -0.121,Y -654.888,Z 850.391,A 0.000,B 0.000,C 90.000,E1 286.315} C_DIS
LIN {X 0.272,Y -656.645,Z 850.388,A 0.000,B 0.000,C 90.000,E1 285.788} C_DIS
LIN {X 0.114,Y -658.867,Z 850.384,A 0.000,B 0.000,C 90.000,E1 285.064} C_DIS
LIN {X -0.097,Y -660.049,Z 850.381,A 0.000,B 0.000,C 90.000,E1 284.592} C_DIS
LIN {X 0.245,Y -661.381,Z 850.377,A 0.000,B 0.000,C 90.000,E1 283.828} C_DIS
LIN {X -0.042,Y -662.351,Z 850.373,A 0.000,B 0.000,C 90.000,E1 283.119} C_DIS
LIN {X -0.230,Y -662.790,Z 850.370,A 0.000,B 0.000,C 90.000,E1 282.647} C_DIS
LIN {X 0.233,Y -663.030,Z 850.367,A 0.000,B 0.000,C 90.000,E1 282.119} C_DIS
LIN {X -0.088,Y -663.010,Z 850.365,A 0.000,B 0.000,C 90.000,E1 281.658} C_DIS
LIN {X 0.283,Y -662.624,Z 850.361,A 0.000,B 0.000,C 90.000,E1 280.894} C_DIS
LIN {X -0.029,Y -662.154,Z 850.358,A 0.000,B 0.000,C 90.000,E1 280.433} C_DIS
LIN {X -0.225,Y -661.465,Z 850.355,A 0.000,B 0.000,C 90.000,E1 279.962} C_DIS
LIN {X 0.112,Y -660.345,Z 850.353,A 0.000,B 0.000,C 90.000,E1 279.443} C_DIS
LIN {X -0.101,Y -658.966,Z 850.350,A 0.000,B 0.000,C 90.000,E1 278.973} C_DIS
LIN {X -0.314,Y -658.182,Z 850.349,A 0.000,B 0.000,C 90.000,E1 278.746} C_DIS
LIN {X 0.104,Y -656.286,Z 850.346,A 0.000,B 0.000,C 90.000,E1 278.219} C_DIS
LIN {X 0.302,Y -653.395,Z 850.342,A 0.000,B 0.000,C 90.000,E1 277.587} C_DIS
LIN {X -0.088,Y -649.917,Z 850.339,A 0.000,B 0.000,C 90.000,E1 277.004} C_DIS
LIN {X 0.215,Y -647.629,Z 850.337,A 0.000,B 0.000,C 90.000,E1 276.606} C_DIS
LIN {X -0.229,Y -643.047,Z 850.333,A 0.000,B 0.000,C 90.000,E1 276.024} C_DIS
LIN {X -0.077,Y -638.737,Z 850.331,A 0.000,B 0.000,C 90.000,E1 275.511} C_DIS
LIN {X 0.233,Y -632.525,Z 850.327,A 0.000,B 0.000,C 90.000,E1 274.878} C_DIS
LIN {X -0.047,Y -625.517,Z 850.324,A 0.000,B 0.000,C 90.000,E1 274.359} C_DIS
LIN {X -0.266,Y -618.086,Z 850.322,A 0.000,B 0.000,C 90.000,E1 273.898} C_DIS
LIN {X 0.094,Y -611.760,Z 850.320,A 0.000,B 0.000,C 90.000,E1 273.498} C_DIS
LIN {X 0.108,Y -604.899,Z 850.318,A 0.000,B 0.000,C 90.000,E1 273.154} C_DIS
LIN {X -0.106,Y -598.194,Z 850.316,A 0.000,B 0.000,C 90.000,E1 272.865} C_DIS
LIN {X -0.065,Y -590.932,Z 850.314,A 0.000,B 0.000,C 90.000,E1 272.579} C_DIS
LIN {X -0.139,Y -585.255,Z 850.313,A 0.000,B 0.000,C 90.000,E1 272.407} C_DIS
LIN {X 0.230,Y -577.362,Z 850.312,A 0.000,B 0.000,C 90.000,E1 272.178} C_DIS
LIN {X -0.044,Y -571.438,Z 850.312,A 0.000,B 0.000,C 90.000,E1 272.121} C_DIS
LIN {X -0.101,Y -564.350,Z 850.311,A 0.000,B 0.000,C 90.000,E1 272.064} C_DIS
LIN {X 0.270,Y -557.293,Z 850.311,A 0.000,B 0.000,C 90.000,E1 272.007} C_DIS
LIN {X 0.005,Y -553.487,Z 850.311,A 0.000,B 0.000,C 90.000,E1 272.007} C_DIS
LIN {X 0.156,Y -551.794,Z 850.311,A 0.000,B 0.000,C 90.000,E1 271.949} C_DIS
LIN {X 0.053,Y -549.818,Z 850.311,A 0.000,B 0.000,C 90.000,E1 271.892} C_DIS
LIN {X 0.018,Y -549.737,Z 850.311,A 0.000,B 0.000,C 90.000,E1 271.892} C_DIS
LIN {X -0.075,Y -548.732,Z 850.310,A 0.000,B 0.000,C 90.000,E1 271.718} C_DIS
LIN {X 0.225,Y -548.159,Z 850.309,A 0.000,B 0.000,C 90.000,E1 271.547} C_DIS
LIN {X 0.009,Y -547.252,Z 850.306,A 0.000,B 0.000,C 90.000,E1 271.146} C_DIS
LIN {X 0.101,Y -546.486,Z 850.303,A 0.000,B 0.000,C 90.000,E1 270.573} C_DIS
LIN {X -0.121,Y -544.611,Z 850.291,A 0.000,B 0.000,C 90.000,E1 268.339} C_DIS
LIN {X 0.122,Y -543.430,Z 850.281,A 0.000,B 0.000,C 90.000,E1 266.617} C_DIS
LIN {X -0.195,Y -542.241,Z 850.272,A 0.000,B 0.000,C 90.000,E1 264.951} C_DIS
LIN {X -0.021,Y -541.219,Z 850.264,A 0.000,B 0.000,C 90.000,E1 263.514} C_DIS
LIN {X -0.282,Y -539.675,Z 850.255,A 0.000,B 0.000,C 90.000,E1 261.837} C_DIS
LIN {X -0.024,Y -538.383,Z 850.247,A 0.000,B 0.000,C 90.000,E1 260.387} C_DIS
LIN {X -0.202,Y -536.455,Z 850.236,A 0.000,B 0.000,C 90.000,E1 258.409} C_DIS
LIN {X 0.202,Y -534.969,Z 850.228,A 0.000,B 0.000,C 90.000,E1 256.937} C_DIS
LIN {X 0.150,Y -532.543,Z 850.216,A 0.000,B 0.000,C 90.000,E1 254.936} C_DIS
LIN {X 0.283,Y -530.548,Z 850.207,A 0.000,B 0.000,C 90.000,E1 253.196} C_DIS
LIN {X -0.123,Y -528.438,Z 850.197,A 0.000,B 0.000,C 90.000,E1 251.511} C_DIS
LIN {X -0.082,Y -526.587,Z 850.189,A 0.000,B 0.000,C 90.000,E1 250.061} C_DIS
LIN {X 0.266,Y -524.215,Z 850.180,A 0.000,B 0.000,C 90.000,E1 248.284} C_DIS
LIN {X -0.092,Y -522.129,Z 850.172,A 0.000,B 0.000,C 90.000,E1 246.869} C_DIS
LIN {X 0.253,Y -520.407,Z 850.165,A 0.000,B 0.000,C 90.000,E1 245.665} C_DIS
LIN {X 0.023,Y -518.084,Z 850.157,A 0.000,B 0.000,C 90.000,E1 244.229} C_DIS
LIN {X 0.199,Y -515.555,Z 850.149,A 0.000,B 0.000,C 90.000,E1 242.743} C_DIS
LIN {X -0.120,Y -512.991,Z 850.141,A 0.000,B 0.000,C 90.000,E1 241.307} C_DIS
LIN {X -0.128,Y -510.911,Z 850.134,A 0.000,B 0.000,C 90.000,E1 240.127} C_DIS
LIN {X 0.054,Y -507.559,Z 850.124,A 0.000,B 0.000,C 90.000,E1 238.329} C_DIS
LIN {X 0.216,Y -505.283,Z 850.117,A 0.000,B 0.000,C 90.000,E1 237.120} C_DIS
LIN {X -0.086,Y -502.747,Z 850.111,A 0.000,B 0.000,C 90.000,E1 235.960} C_DIS
LIN {X -0.262,Y -499.444,Z 850.103,A 0.000,B 0.000,C 90.000,E1 234.482} C_DIS
LIN {X -0.059,Y -493.018,Z 850.087,A 0.000,B 0.000,C 90.000,E1 231.743} C_DIS
LIN {X 0.189,Y -489.422,Z 850.079,A 0.000,B 0.000,C 90.000,E1 230.194} C_DIS
LIN {X -0.154,Y -486.584,Z 850.072,A 0.000,B 0.000,C 90.000,E1 229.013} C_DIS
LIN {X -0.088,Y -483.111,Z 850.064,A 0.000,B 0.000,C 90.000,E1 227.472} C_DIS
LIN {X -0.190,Y -478.393,Z 850.052,A 0.000,B 0.000,C 90.000,E1 225.324} C_DIS
LIN {X 0.272,Y -475.817,Z 850.045,A 0.000,B 0.000,C 90.000,E1 224.028} C_DIS
LIN {X -0.033,Y -471.081,Z 850.033,A 0.000,B 0.000,C 90.000,E1 221.881} C_DIS
LIN {X -0.145,Y -467.016,Z 850.022,A 0.000,B 0.000,C 90.000,E1 220.011} C_DIS
LIN {X 0.260,Y -463.700,Z 850.013,A 0.000,B 0.000,C 90.000,E1 218.382} C_DIS
LIN {X 0.169,Y -461.755,Z 850.008,A 0.000,B 0.000,C 90.000,E1 217.443} C_DIS
LIN {X 0.168,Y -459.151,Z 850.001,A 0.000,B 0.000,C 90.000,E1 216.171} C_DIS
LIN {X -0.035,Y -455.004,Z 849.990,A 0.000,B 0.000,C 90.000,E1 214.278} C_DIS
LIN {X 0.208,Y -449.473,Z 849.976,A 0.000,B 0.000,C 90.000,E1 211.671} C_DIS
LIN {X 0.052,Y -445.351,Z 849.965,A 0.000,B 0.000,C 90.000,E1 209.745} C_DIS
LIN {X 0.184,Y -441.368,Z 849.954,A 0.000,B 0.000,C 90.000,E1 207.769} C_DIS
LIN {X -0.193,Y -437.351,Z 849.943,A 0.000,B 0.000,C 90.000,E1 205.848} C_DIS
LIN {X 0.122,Y -434.017,Z 849.934,A 0.000,B 0.000,C 90.000,E1 204.155} C_DIS
LIN {X -0.029,Y -430.636,Z 849.925,A 0.000,B 0.000,C 90.000,E1 202.514} C_DIS
LIN {X 0.177,Y -426.708,Z 849.914,A 0.000,B 0.000,C 90.000,E1 200.482} C_DIS
LIN {X -0.214,Y -422.145,Z 849.901,A 0.000,B 0.000,C 90.000,E1 198.181} C_DIS
END
